// TIA Portal V20 program export: 6 tag tables, 4 data types, 72 data blocks, 38 code blocks (in call order from the OBs), 73 instance data blocks

VAR_GLOBAL   // PLC tag table "06_ProductionData"
END_VAR
VAR_GLOBAL CONSTANT   // user constants
   NO_DATASETS_CYCLETIMER : Int := 8;   // SICAR: Anzahl Datensätze Taktzeiten / SICAR: Number of data sets Cycle Timer
   NO_DATASETS_LIMITVALUES : Int := 1;   // SICAR: Anzahl Datensätze Grenzwerte / SICAR: Number of data sets Limit Value
   NO_DATASETS_SHIFTCOUNTER : Int := 1;   // SICAR: Anzahl Datensätze Schichtzähler / SICAR: Number of data sets Shift Counter
   NO_DATASETS_COUNTER : Int := 1;   // SICAR: Anzahl Datensätze Zähler / SICAR: Number of data sets Counter
END_VAR

VAR_GLOBAL   // PLC tag table "07_Energy"
   PAC3220InPut AT %I500.0 : "LER_typePAC3220Input_Status";
   "Active energy import tariff 1(F)" AT %ID612 : Real;
   "Reactive energy import tariff 1 (F)" AT %ID616 : Real;
   "Apparent energy tariff 1 (F)" AT %ID620 : Real;
   "Active energy export tariff 1(F)" AT %ID624 : Real;
   "Reactive energy export tariff 1 (F)" AT %ID628 : Real;
   "Apparent power L1" AT %ID632 : Real;
   "Apparent power L2" AT %ID636 : Real;
   "Apparent power L3" AT %ID640 : Real;
   "Active power L1" AT %ID644 : Real;
   "Active power L2" AT %ID648 : Real;
   "Active power L3" AT %ID652 : Real;
   "Reactive power L1" AT %ID656 : Real;
   "Reactive power L2" AT %ID660 : Real;
   "Reactive power L3" AT %ID664 : Real;
   PAC3220OutPut AT %Q500.0 : "LER_typePAC3220Output_Status";
END_VAR
VAR_GLOBAL CONSTANT   // user constants
   NO_OF_MACHINES : USInt := 1;   // SICAR: No of machines for EE-Monitor
   NO_OF_MEASUREPOINTS : USInt := 1;   // SICAR: Anzahl der Messstellen für EE-Monitor / SICAR: No of measurepoints for EE-Monitor
   "DP_FRWA1_1_0_000CC1-KE50~DP_FRWA1_1_0_000CC1-KE50_900" : Hw_Io := 10;
END_VAR

VAR_GLOBAL   // PLC tag table "08_CmInfo"
END_VAR
VAR_GLOBAL CONSTANT   // user constants
   NO_OF_RF_IDENT_DEVICES : USInt := 0;   // SICAR: Anzahl der RF Lesestellen / SICAR: Number of RF readers
   NO_OF_RF_ANTENNA_DEVICES : USInt := 2;   // SICAR: Number of RF antennas
END_VAR

VAR_GLOBAL   // PLC tag table "11_Settings"
END_VAR
VAR_GLOBAL CONSTANT   // user constants
   MAX_NO_OF_DEVICES_IRT : Int := 200;
   MAX_NO_OF_MODULES_IRT : Int := 200;
   MAX_NO_OF_DEVICES_RT : Int := 200;
   MAX_NO_OF_MODULES_RT : Int := 200;
END_VAR

VAR_GLOBAL   // PLC tag table "CentralFunctions"
END_VAR
VAR_GLOBAL CONSTANT   // user constants
   MAX_NO_OF_DEVICES_X1 : Int := 100;
   MAX_NO_OF_MODULES_X1 : Int := 100;
   MAX_NO_OF_DEVICES_X2 : Int := 100;
   MAX_NO_OF_MODULES_X2 : Int := 100;
END_VAR

VAR_GLOBAL   // PLC tag table "TextListId"
END_VAR
VAR_GLOBAL CONSTANT   // user constants
   TEXT_LIST_ID_PN_DEV_DIAG : Int := 591;   // SICAR: ID von SPS Alarm Textlist / SICAR: ID of PLC Alarm text list
   TEXT_LIST_ID_CHECKSUM : Int := 584;   // SICAR: ID von SPS Alarm Textlist / SICAR: ID of PLC Alarm text list
   TEXT_LIST_ID_EEEMONITOR_REPORT : Int := 562;   // SICAR: ID von SPS Alarm Textlist / SICAR: ID of PLC Alarm text list
   TEXT_LIST_ID_EEEMONITOR_CALC : Int := 561;   // SICAR: ID von SPS Alarm Textlist / SICAR: ID of PLC Alarm text list
   TEXT_LIST_ID_IDENT_SYSTEM : Int := 516;   // SICAR: ID of PLC Alarm for ident demo
   TEXT_LIST_ID_SMC_PD : Int := 585;   // SICAR: ID von SPS Alarm Textlist / SICAR: ID of PLC Alarm text list
   TEXT_LIST_ID_MOTORSTARTERS : Int := 588;   // SICAR: ID of PLC Alarm for motorstarter Demo
   TEXT_LIST_ID_DEV_FWD_REV : Int := 592;   // SICAR: ID of PLC Alarm for motorstarter Demo
END_VAR

TYPE "typeReelCutToStack"
   STRUCT
      Load_Enable : Bool;
      Load_Complete_Comfirm : Bool;
      Cell_Data_Report : Bool;
      signal3 : Bool;
      signal4 : Bool;
      signal5 : Bool;
      signal6 : Bool;
      signal7 : Bool;
      signal8 : Bool;
      signal9 : Bool;
      signal10 : Bool;
      signal11 : Bool;
      signal12 : Bool;
      signal13 : Bool;
      signal14 : Bool;
      HeartBeat : Bool;
      signal16 : Bool;
      signal17 : Bool;
      signal18 : Bool;
      signal19 : Bool;
      signal20 : Bool;
      signal21 : Bool;
      signal22 : Bool;
      signal23 : Bool;
      signal24 : Bool;
      signal25 : Bool;
      signal26 : Bool;
      signal27 : Bool;
      signal28 : Bool;
      signal29 : Bool;
      signal30 : Bool;
      signal31 : Bool;
      signal32 : Bool;
      signal33 : Bool;
      signal34 : Bool;
      signal35 : Bool;
      signal36 : Bool;
      signal37 : Bool;
      signal38 : Bool;
      signal39 : Bool;
      signal40 : Bool;
      signal41 : Bool;
      signal42 : Bool;
      signal43 : Bool;
      signal44 : Bool;
      signal45 : Bool;
      signal46 : Bool;
      signal47 : Bool;
      signal48 : Bool;
      signal49 : Bool;
      signal50 : Bool;
      signal51 : Bool;
      signal52 : Bool;
      signal53 : Bool;
      signal54 : Bool;
      signal55 : Bool;
      signal56 : Bool;
      signal57 : Bool;
      signal58 : Bool;
      signal59 : Bool;
      signal60 : Bool;
      signal61 : Bool;
      signal62 : Bool;
      signal63 : Bool;
      signal64 : Bool;
      signal65 : Bool;
      signal66 : Bool;
      signal67 : Bool;
      signal68 : Bool;
      signal69 : Bool;
      signal70 : Bool;
      signal71 : Bool;
      signal72 : Bool;
      signal73 : Bool;
      signal74 : Bool;
      signal75 : Bool;
      signal76 : Bool;
      signal77 : Bool;
      signal78 : Bool;
      signal79 : Bool;
      signal80 : Bool;
      signal81 : Bool;
      signal82 : Bool;
      signal83 : Bool;
      signal84 : Bool;
      signal85 : Bool;
      signal86 : Bool;
      signal87 : Bool;
      signal88 : Bool;
      signal89 : Bool;
      signal90 : Bool;
      signal91 : Bool;
      signal92 : Bool;
      signal93 : Bool;
      signal94 : Bool;
      signal95 : Bool;
   END_STRUCT;
END_TYPE

TYPE "typeStackToReelCut"
   STRUCT
      Load_Requset : Bool;
      Load_Busy : Bool;
      Load_Complete : Bool;
      Cell_Data_Request : Bool;
      Cell_Data_Report_Ack : Bool;
      Cell_Data_Report_Nck : Bool;
      signal6 : Bool;
      signal7 : Bool;
      signal8 : Bool;
      signal9 : Bool;
      signal10 : Bool;
      signal11 : Bool;
      signal12 : Bool;
      signal13 : Bool;
      signal14 : Bool;
      HeartBeat : Bool;
      signal16 : Bool;
      signal17 : Bool;
      signal18 : Bool;
      signal19 : Bool;
      signal20 : Bool;
      signal21 : Bool;
      signal22 : Bool;
      signal23 : Bool;
      signal24 : Bool;
      signal25 : Bool;
      signal26 : Bool;
      signal27 : Bool;
      signal28 : Bool;
      signal29 : Bool;
      signal30 : Bool;
      signal31 : Bool;
      signal32 : Bool;
      signal33 : Bool;
      signal34 : Bool;
      signal35 : Bool;
      signal36 : Bool;
      signal37 : Bool;
      signal38 : Bool;
      signal39 : Bool;
      signal40 : Bool;
      signal41 : Bool;
      signal42 : Bool;
      signal43 : Bool;
      signal44 : Bool;
      signal45 : Bool;
      signal46 : Bool;
      signal47 : Bool;
      signal48 : Bool;
      signal49 : Bool;
      signal50 : Bool;
      signal51 : Bool;
      signal52 : Bool;
      signal53 : Bool;
      signal54 : Bool;
      signal55 : Bool;
      signal56 : Bool;
      signal57 : Bool;
      signal58 : Bool;
      signal59 : Bool;
      signal60 : Bool;
      signal61 : Bool;
      signal62 : Bool;
      signal63 : Bool;
      signal64 : Bool;
      signal65 : Bool;
      signal66 : Bool;
      signal67 : Bool;
      signal68 : Bool;
      signal69 : Bool;
      signal70 : Bool;
      signal71 : Bool;
      signal72 : Bool;
      signal73 : Bool;
      signal74 : Bool;
      signal75 : Bool;
      signal76 : Bool;
      signal77 : Bool;
      signal78 : Bool;
      signal79 : Bool;
      signal80 : Bool;
      signal81 : Bool;
      signal82 : Bool;
      signal83 : Bool;
      signal84 : Bool;
      signal85 : Bool;
      signal86 : Bool;
      signal87 : Bool;
      signal88 : Bool;
      signal89 : Bool;
      signal90 : Bool;
      signal91 : Bool;
      signal92 : Bool;
      signal93 : Bool;
      signal94 : Bool;
      signal95 : Bool;
   END_STRUCT;
END_TYPE

TYPE "typeIdentRf"
// stored: Access Published
   STRUCT
      IdentRfAntena : Array[0.."NO_OF_RF_ANTENNA_DEVICES"] of "LSicar_typeIdentInterfaceHmi";
   END_STRUCT;
END_TYPE

TYPE "typeIdentRfHmi"
// stored: Access Published
   STRUCT
      selectedRfReader : USInt;   // Reader ID
      selectedAntena : USInt;
      rfReaderId : USInt;   // RF Reader ID
      numberOfRf : USInt;   // Anzahl der RFID Antriebe / Number of used RFIDs
      rfReader : "LSicar_typeIdentInterfaceHmi";   // RF Reader
   END_STRUCT;
END_TYPE

DATA_BLOCK "Hmi"   // DB4
// stored: MemoryReserve 100
   VAR
      mainHeader : Array[0.."NO_OF_PANELS"] of "LAF_typeHeader";   // Input from the status bar of the HMI
      operationInterlock : "LAF_typeOperationInterlockInterface";
   END_VAR
BEGIN
   mainHeader[0].plcToHmi.modeRequestsButtons.visibility := 16#0;
   mainHeader[0].plcToHmi.specialFunctionButtons.visibility := 16#0071_FFFF;
   mainHeader[0].plcToHmi.specialFunctionButtons.operatorControlAllowed := 16#0;
   mainHeader[0].plcToHmi.specialFunctionButtons.active := 16#0;
END_DATA_BLOCK

DATA_BLOCK "LRemoteAccess_Data"   // DB275
TITLE = Data
AUTHOR : Siemens
// Storing data about mobile panel and UCP connection status
// stored: MemoryReserve 100
   VAR
      mobilePanel1 : "LRemoteAccess_typeMobilePanel";
      connectionBoxes : Array[1..2] of "LRemoteAccess_typeConnectionBox";
      ActivationMobileDP { S7_SetPoint := 'True'} : "LRemoteAccess_typeMobile_DeActivate";   // Activate Mobile Panel
      DeactivationMobileDP { S7_SetPoint := 'True'} : "LRemoteAccess_typeMobile_DeActivate";   // Deactivate Mobile Panel
      connectionTimeout { S7_SetPoint := 'True'} : Time := T#5s;   // Connection timeout. Keep greater than 3 sec. Default 5 sec.
   END_VAR
BEGIN
   connectionBoxes[1].ID := 14;
   connectionBoxes[2].ID := 15;
END_DATA_BLOCK

DATA_BLOCK "Simulation"   // DB134
TITLE = Simulation
// Simulation data
// stored: MemoryReserve 100
   VAR
      data : "LAF_typeSimulation";
      hmiSimulationAxis { S7_SetPoint := 'True'} : Array[0..10] of LReal;
   END_VAR
BEGIN
END_DATA_BLOCK

DATA_BLOCK "HMI_Interface_Overview"   // DB276
// stored: Access Published, MemoryReserve 100
   VAR
      State : Struct
         "Anode Reel Cut" : "HMI_IF_OverView_Unit_UDT";
         "Cathode Reel Cut" : "HMI_IF_OverView_Unit_UDT";
         "Stacker #1" : "HMI_IF_OverView_Unit_UDT";
         "Stacker #2" : "HMI_IF_OverView_Unit_UDT";
         Inspection : "HMI_IF_OverView_Unit_UDT";
      END_STRUCT;
   END_VAR
BEGIN
END_DATA_BLOCK

DATA_BLOCK "LAF_InternalManual"   // DB43
VERSION : 19.0
// stored: MemoryReserve 100
   VAR
      hmi : Array[1..1] of "LAF_typeManHmiDisp";   // Anzahl der HMIs - modifizieren Sie die Array-Größe auf Basis der erforderlichen HMI / number of HMIs - modify the array size based on the required HMIs / número de HMI: modificar el tamaño del array según las HMI requeridas / nombre d'IHM - modifier la taille du tableau en fonction du nombre d'IHM requis / numero di HMI - modificare la dimensione di array in base alle HMI richieste / HMI 수 - 필요한 HMI에 따라 배열 크기를 수정합니다. / HMI 数量 - 根据所需的 HMI 修改数组大小
      manualOperationEnabled : Bool;   // feedback whether the manual operation lines are selected
      emsWithManualOpConfigured { ExternalWritable := 'False'} : "LGM_emsWithManualOpConfigured";   // List of EMs with manual operation configured, for HMI button visibility
      disableUnit1 { S7_SetPoint := 'True'} : Bool;
      RisingEdge : Bool;
   END_VAR
BEGIN
END_DATA_BLOCK

DATA_BLOCK "ManualOperationControl_Template"   // DB91
// stored: MemoryReserve 100
   VAR
      manualOperationEm { ExternalAccessible := 'False'; ExternalVisible := 'False'; ExternalWritable := 'False'} : "LAF_typeManEm";
      manualOperationEmArea { ExternalAccessible := 'False'; ExternalVisible := 'False'; ExternalWritable := 'False'} : Array[1..1] of "LAF_typeManOperationArea";
      manualOperationCms { ExternalAccessible := 'False'; ExternalVisible := 'False'; ExternalWritable := 'False'} : Array[1..1] of "LAF_typeManOperation";
   END_VAR
BEGIN
   manualOperationEm.equipmentModuleNum := 3400;
END_DATA_BLOCK

DATA_BLOCK "OperatorPrompts"   // DB123
// stored: Access Published, MemoryReserve 100
   VAR
      triggers { ExternalAccessible := 'False'; ExternalVisible := 'False'; ExternalWritable := 'False'} : Array[1..63] of Bool;
      activeOperatorPrompt { ExternalWritable := 'False'} : Int;
      ack : Bool;
   END_VAR
BEGIN
END_DATA_BLOCK

DATA_BLOCK "ProdDataInterfaceHmi"   // DB53
TITLE = HMI und Anwender Schnittstelle für Produktionsdaten / HMI and user interface for production data
AUTHOR : SICAR
FAMILY : ProdData
// FUNKTIONSBESCHREIBUNG: 
// Der Baustein beinhaltet alle Informationen zum und vom HMI, sowie die Anwenderschnittstellen für die Produktionsdaten
// Weitere Hinweise: siehe SICAR anwenderdefinierte Dokumentation / SICAR Online-Hilfe.
// DESCRIPTION OF FUNCTIONS:
// stored: MemoryReserve 100
   VAR RETAIN
      numberOfDataSets : "LSicar_typeNumberOfDataSets";   // Anzahl konfigurierter Datensätze / Number of configured data sets
   END_VAR
   VAR
      colorCodeLimitSummary : UInt;   // Gesamt Status Grenzwerte / Overall status Limit values
      colorCodeLimitSelButton : Array[0..8] of UInt;   // Farbcode für Datensatz Anwahl Button (Grenzwerte) / Color code for data set select button (Limit values)
   END_VAR
   VAR RETAIN
      counterDataSetSel : Int := 1;   // Angewählter Datensatz Zaehler / selected data set counter
      counterDataSet : Array[0.."NO_DATASETS_COUNTER"] of "LSicar_typeCounter";   // Datensätze Zähler / Data sets counter
      cycleTimerDataSetSel : Int := 1;   // Angewaehlter Datensatz Taktzeiten / selected data set cycle timer
      cycleTimerDataSet : Array[0.."NO_DATASETS_CYCLETIMER"] of "LSicar_typeCycleTimer";   // Datensätze Taktzeiten / Data sets cycle timer
      limitValueDataSetSel : Int := 1;   // Angwaehlter Datensatz Grenzwerte / selected data set limit values
      limitDataSet : Array[0.."NO_DATASETS_LIMITVALUES"] of "LSicar_typeLimitValue";   // Datensätze Grenzwerte / Data sets limit .values
      shiftCounterDataSetSel : Int := 1;   // Angewaehlter Datensatz Schichtzaehler / selected data set shift counter
      shiftCounterDataSet : Array[0.."NO_DATASETS_SHIFTCOUNTER"] of "LSicar_typeShiftCounter";   // Datensätze Schichtzähler / Data sets shift counter
      shiftCountOeeDataSetSel : Int := 1;   // Angewaehlter Datensatz OEE / selected data set OEE
      shiftCounterOeeDataSet : Array[0.."NO_DATASETS_SHIFTCOUNTER"] of "LSicar_typeShiftCounterOee";   // Datensätze Schichtzähler OEE / Data sets shift counter OEE
   END_VAR
BEGIN
END_DATA_BLOCK

DATA_BLOCK "ProdDataSimulation"   // DB5
{ DB_Accessible_From_OPC_UA := 'FALSE' }
// stored: DBAccessibleFromOPCUA false, DBAccessibleFromWebserver false, MemoryReserve 100
   VAR
      ProdDataCounter { ExternalAccessible := 'False'; ExternalVisible := 'False'; ExternalWritable := 'False'} : Struct   // Test tag prod data
         ProdDataCounter1Up1 : Bool;   // Test Variable Prod. Daten / Test tag prod data
         ProdDataCounter1Up2 : Bool;   // Test Variable Prod. Daten / Test tag prod data
         ProdDataCounter1Down1 : Bool;   // Test Variable Prod. Daten / Test tag prod data
         ProdDataCounter1Down2 : Bool;   // Test Variable Prod. Daten / Test tag prod data
         ProdDataCounter1Reset1 : Bool;   // Test Variable Prod. Daten / Test tag prod data
         ProdDataCounter1Reset2 : Bool;   // Test Variable Prod. Daten / Test tag prod data
         ProdDataCounter1ResetAll : Bool;   // Test Variable Prod. Daten / Test tag prod data
         ProdDataCounter2Up1 : Bool;
         ProdDataCounter2Up2 : Bool;
         ProdDataCounter2Down1 : Bool;
         ProdDataCounter2Down2 : Bool;
         ProdDataCounter2Reset1 : Bool;
         ProdDataCounter2Reset2 : Bool;
         ProdDataCounter2ResetAll : Bool;
         userInterfaceVisibilityDataSet1Counter : DWord := 2#0000_0000_0000_0000_0000_0000_0011_1111;
         userInterfaceVisibilityDataSet2Counter : DWord := 2#0000_0000_0000_1111_1111_1111_1111_1111;
         ProdDataEnable : Bool;
      END_STRUCT;
      ProdDataCyclic { ExternalAccessible := 'False'; ExternalVisible := 'False'; ExternalWritable := 'False'} : Struct   // Test tag prod data
         cycleTimer1Run1 : Bool;   // Test Variable Prod. Daten / Test tag prod data
         cycleTimer1Run2 : Bool;   // Test Variable Prod. Daten / Test tag prod data
         cycleTimer1Hold1 : Bool;   // Test Variable Prod. Daten / Test tag prod data
         cycleTimer1Hold2 : Bool;   // Test Variable Prod. Daten / Test tag prod data
         cycleTimer1Reset1 : Bool;   // Test Variable Prod. Daten / Test tag prod data
         cycleTimer1Reset2 : Bool;   // Test Variable Prod. Daten / Test tag prod data
         cycleTimer1ResetAll : Bool;   // Test Variable Prod. Daten / Test tag prod data
         cycleTimer2Run1 : Bool;   // Test Variable Prod. Daten / Test tag prod data
         cycleTimer2Run2 : Bool;   // Test Variable Prod. Daten / Test tag prod data
         cycleTimer2Hold1 : Bool;   // Test Variable Prod. Daten / Test tag prod data
         cycleTimer2Hold2 : Bool;   // Test Variable Prod. Daten / Test tag prod data
         cycleTimer2Reset1 : Bool;   // Test Variable Prod. Daten / Test tag prod data
         cycleTimer2Reset2 : Bool;   // Test Variable Prod. Daten / Test tag prod data
         cycleTimer2ResetAll : Bool;   // Test Variable Prod. Daten / Test tag prod data
         cyclicTimerEnable : Bool;
         userInterfaceVisibilityDataSet1Cyclic : DWord := 2#0000_0000_0000_0000_0000_0000_0000_1111;
         userInterfaceVisibilityDataSet2Cyclic : DWord := 2#0000_0000_0000_0000_0000_0000_0000_1111;
         userInterfaceVisibilityDataSet3Cyclic : DWord := 2#0000_0000_0000_1000_0111_1111_1101_1111;
         userInterfaceVisibilityDataSet4Cyclic : DWord := 2#0000_0000_0000_0000_0000_0000_1111_1111;
         userInterfaceVisibilityDataSet5Cyclic : DWord := 2#0000_0000_0000_0000_0000_0000_0000_0001;
         userInterfaceVisibilityDataSet6Cyclic : DWord := 2#0000_0000_0000_0000_0000_0000_0000_0111;
         userInterfaceVisibilityDataSet7Cyclic : DWord := 2#0000_0000_0000_0000_0011_1100_0000_0111;
         userInterfaceVisibilityDataSet8Cyclic : DWord := 2#0000_0000_0000_1111_1111_1100_1111_1111;
      END_STRUCT;
      ProdDataLimitValues { ExternalAccessible := 'False'; ExternalVisible := 'False'; ExternalWritable := 'False'} : Struct   // Test tag prod data
         limitVal1Count1PreWarn1 : Bool;   // Test Variable Prod. Daten / Test tag prod data
         limitVal1Count1PreWarn3 : Bool;   // Test Variable Prod. Daten / Test tag prod data
         limitVal1Count1PreWarn2 : Bool;   // Test Variable Prod. Daten / Test tag prod data
         limitVal1Count1Alarm1 : Bool;   // Test Variable Prod. Daten / Test tag prod data
         limitVal1Count1Alarm3 : Bool;   // Test Variable Prod. Daten / Test tag prod data
         limitVal1Count1Alarm2 : Bool;   // Test Variable Prod. Daten / Test tag prod data
         limitVal1Count1 : Bool;   // Test Variable Prod. Daten / Test tag prod data
         limitVal1Count2 : Bool;   // Test Variable Prod. Daten / Test tag prod data
         limitVal1Count3 : Bool;   // Test Variable Prod. Daten / Test tag prod data
         limitVal1Set1 : Bool;   // Test Variable Prod. Daten / Test tag prod data
         limitVal1Set3 : Bool;   // Test Variable Prod. Daten / Test tag prod data
         limitVal1Set2 : Bool;   // Test Variable Prod. Daten / Test tag prod data
         limitValuesEnable : Bool;
         userInterfaceVisibilityDataSet2LimitValues : DWord := 2#0000_0000_0000_0000_0000_0011_1111_1111;
         userInterfaceVisibilityDataSet1LimitValues : DWord := 2#0000_0000_0000_0000_0000_0000_0000_1111;
      END_STRUCT;
      ProdDataShiftCounter { ExternalAccessible := 'False'; ExternalVisible := 'False'; ExternalWritable := 'False'} : Struct   // Test tag prod data
         shiftCounter1Cnt1Curr : Bool;   // Test Variable Prod. Daten / Test tag prod data
         shiftCounter1Cnt1CurrOk : Bool;   // Test Variable Prod. Daten / Test tag prod data
         shiftCounter1Cnt2Curr : Bool;   // Test Variable Prod. Daten / Test tag prod data
         shiftCounter1Cnt2CurrOk : Bool;   // Test Variable Prod. Daten / Test tag prod data
         shiftCounter1Cnt3Curr : Bool;   // Test Variable Prod. Daten / Test tag prod data
         shiftCounter1Cnt3CurrOk : Bool;   // Test Variable Prod. Daten / Test tag prod data
         shiftCounter1ResetAllExt : Bool;   // Test Variable Prod. Daten / Test tag prod data
         ShiftCounterEnable : Bool;
         userInterfaceVisibilityDataSet2ShiftCounter : DWord := 2#0000_0000_0000_0000_0000_0011_1111_1111;
         userInterfaceVisibilityDataSet1ShiftCounter : DWord := 2#0000_0000_0000_0000_0000_0000_0000_1111;
      END_STRUCT;
      ProdDataShiftCounterOEE { ExternalAccessible := 'False'; ExternalVisible := 'False'; ExternalWritable := 'False'} : Struct   // Test tag prod data
         ShiftCounterOEEEnable : Bool;
         userInterfaceVisibilityDataSet2ShiftCounterOEE : DWord := 2#0000_0000_0000_0000_0000_0011_1111_1111;
         userInterfaceVisibilityDataSet1ShiftCounterOEE : DWord := 2#0000_0000_0000_0000_0000_0000_0000_1111;
      END_STRUCT;
   END_VAR
BEGIN
END_DATA_BLOCK

DATA_BLOCK "ShiftInitBools"   // DB257
// stored: MemoryReserve 100
   VAR
      earlyShift : Bool;
      lateShift : Bool;
      nightShift : Bool;
   END_VAR
BEGIN
END_DATA_BLOCK

DATA_BLOCK "ShiftTimesList"   // DB52
TITLE = Shifttimes / Shift times
{ DB_Accessible_From_OPC_UA := 'FALSE' }
AUTHOR : SICAR
FAMILY : Shiftmodel
// Schichtzeiten Liste / Shift times List
// stored: DBAccessibleFromOPCUA false, MemoryReserve 100
   VAR
      list { ExternalAccessible := 'False'; ExternalVisible := 'False'; ExternalWritable := 'False'} : Array[0..10] of "LSicar_typeShiftmodTime1DaySel";   // Schichtmodel Liste / Shiftmodel list
   END_VAR
BEGIN
   list[3].listValidFor.sunday := TRUE;
   list[4].listValidFor.sunday := FALSE;
   list[1..3].listValidFor.monday := TRUE;
   list[4].listValidFor.monday := FALSE;
   list[1..3].listValidFor.tuesday := TRUE;
   list[4].listValidFor.tuesday := FALSE;
   list[1..3].listValidFor.wednesday := TRUE;
   list[4].listValidFor.wednesday := FALSE;
   list[1..3].listValidFor.thursday := TRUE;
   list[4].listValidFor.thursday := FALSE;
   list[1].listValidFor.friday := TRUE;
   list[3].listValidFor.friday := TRUE;
   list[4].listValidFor.friday := FALSE;
   list[3].listValidFor.saturday := TRUE;
   list[4].listValidFor.saturday := FALSE;
   list[1].shift[1].endCircuitTime := TOD#05:57:00;
   list[1].shift[2].endCircuitTime := TOD#13:57:00;
   list[1].shift[3].endCircuitTime := TOD#21:57:00;
   list[2].shift[1].endCircuitTime := TOD#04:57:00;
   list[2].shift[2].endCircuitTime := TOD#14:27:00;
   list[3].shift[1].endCircuitTime := TOD#05:57:00;
   list[3].shift[2].endCircuitTime := TOD#14:27:00;
   list[3].shift[3].endCircuitTime := TOD#22:57:00;
   list[4].shift[1..3].endCircuitTime := TOD#00:00:00;
   list[1].shift[1].start := TOD#06:00:00;
   list[1].shift[2].start := TOD#14:00:00;
   list[1].shift[3].start := TOD#22:00:00;
   list[2].shift[1].start := TOD#05:00:00;
   list[2].shift[2].start := TOD#14:30:00;
   list[3].shift[1].start := TOD#06:00:00;
   list[3].shift[2].start := TOD#14:30:00;
   list[3].shift[3].start := TOD#23:00:00;
   list[4].shift[1..3].start := TOD#00:00:00;
   list[1].shift[1].break[1].start := TOD#08:00:00;
   list[1].shift[1].break[2].start := TOD#10:00:00;
   list[1].shift[1].break[3].start := TOD#12:00:00;
   list[1].shift[1].break[4].start := TOD#00:00:00;
   list[1].shift[2].break[1].start := TOD#16:00:00;
   list[1].shift[2].break[2].start := TOD#18:00:00;
   list[1].shift[2].break[3].start := TOD#20:00:00;
   list[1].shift[3].break[1].start := TOD#00:00:00;
   list[1].shift[3].break[2].start := TOD#02:00:00;
   list[1].shift[3].break[3].start := TOD#04:00:00;
   list[2].shift[1].break[1].start := TOD#07:00:00;
   list[2].shift[1].break[2].start := TOD#09:00:00;
   list[2].shift[1].break[3].start := TOD#11:00:00;
   list[2].shift[1].break[4].start := TOD#13:00:00;
   list[2].shift[2].break[1].start := TOD#16:30:00;
   list[2].shift[2].break[2].start := TOD#18:30:00;
   list[2].shift[2].break[3].start := TOD#20:30:00;
   list[2].shift[2].break[4].start := TOD#22:00:00;
   list[3].shift[1].break[1].start := TOD#08:00:00;
   list[3].shift[1].break[2].start := TOD#10:00:00;
   list[3].shift[1].break[3].start := TOD#11:30:00;
   list[3].shift[1].break[4].start := TOD#12:30:00;
   list[3].shift[2].break[1].start := TOD#16:00:00;
   list[3].shift[2].break[2].start := TOD#18:00:00;
   list[3].shift[2].break[3].start := TOD#19:30:00;
   list[3].shift[2].break[4].start := TOD#20:30:00;
   list[3].shift[3].break[1].start := TOD#00:00:00;
   list[3].shift[3].break[2].start := TOD#02:00:00;
   list[3].shift[3].break[3].start := TOD#03:30:00;
   list[3].shift[3].break[4].start := TOD#04:30:00;
   list[4].shift[1].break[1..4].start := TOD#00:00:00;
   list[4].shift[2].break[1..4].start := TOD#00:00:00;
   list[4].shift[3].break[1..4].start := TOD#00:00:00;
   list[1].shift[1].break[1].startCircuitTime := TOD#08:02:00;
   list[1].shift[1].break[2].startCircuitTime := TOD#00:00:00;
   list[1].shift[1].break[3].startCircuitTime := TOD#12:02:00;
   list[1].shift[1].break[4].startCircuitTime := TOD#00:00:00;
   list[1].shift[2].break[1].startCircuitTime := TOD#16:02:00;
   list[1].shift[2].break[2].startCircuitTime := TOD#00:00:00;
   list[1].shift[2].break[3].startCircuitTime := TOD#20:02:00;
   list[1].shift[3].break[1].startCircuitTime := TOD#00:02:00;
   list[1].shift[3].break[2].startCircuitTime := TOD#00:00:00;
   list[1].shift[3].break[3].startCircuitTime := TOD#04:02:00;
   list[2].shift[1].break[1].startCircuitTime := TOD#07:02:00;
   list[2].shift[1].break[2].startCircuitTime := TOD#00:00:00;
   list[2].shift[1].break[3].startCircuitTime := TOD#11:02:00;
   list[2].shift[1].break[4].startCircuitTime := TOD#13:02:00;
   list[2].shift[2].break[1].startCircuitTime := TOD#16:32:00;
   list[2].shift[2].break[2].startCircuitTime := TOD#00:00:00;
   list[2].shift[2].break[3].startCircuitTime := TOD#20:32:00;
   list[2].shift[2].break[4].startCircuitTime := TOD#22:02:00;
   list[3].shift[1].break[1].startCircuitTime := TOD#00:00:00;
   list[3].shift[1].break[2].startCircuitTime := TOD#10:02:00;
   list[3].shift[1].break[3].startCircuitTime := TOD#00:00:00;
   list[3].shift[1].break[4].startCircuitTime := TOD#12:32:00;
   list[3].shift[2].break[1].startCircuitTime := TOD#00:00:00;
   list[3].shift[2].break[2].startCircuitTime := TOD#18:02:00;
   list[3].shift[2].break[3].startCircuitTime := TOD#00:00:00;
   list[3].shift[2].break[4].startCircuitTime := TOD#20:32:00;
   list[3].shift[3].break[1].startCircuitTime := TOD#00:00:00;
   list[3].shift[3].break[2].startCircuitTime := TOD#02:02:00;
   list[3].shift[3].break[3..4].startCircuitTime := TOD#00:00:00;
   list[4].shift[1].break[1..4].startCircuitTime := TOD#00:00:00;
   list[4].shift[2].break[1..4].startCircuitTime := TOD#00:00:00;
   list[4].shift[3].break[1..4].startCircuitTime := TOD#00:00:00;
   list[1].shift[1].break[1].endCircuitTime := TOD#08:13:00;
   list[1].shift[1].break[2].endCircuitTime := TOD#00:00:00;
   list[1].shift[1].break[3].endCircuitTime := TOD#12:13:00;
   list[1].shift[1].break[4].endCircuitTime := TOD#00:00:00;
   list[1].shift[2].break[1].endCircuitTime := TOD#16:13:00;
   list[1].shift[2].break[2].endCircuitTime := TOD#00:00:00;
   list[1].shift[2].break[3].endCircuitTime := TOD#20:13:00;
   list[1].shift[3].break[1].endCircuitTime := TOD#00:13:00;
   list[1].shift[3].break[2].endCircuitTime := TOD#00:00:00;
   list[1].shift[3].break[3].endCircuitTime := TOD#04:13:00;
   list[2].shift[1].break[1].endCircuitTime := TOD#07:13:00;
   list[2].shift[1].break[2].endCircuitTime := TOD#00:00:00;
   list[2].shift[1].break[3].endCircuitTime := TOD#11:13:00;
   list[2].shift[1].break[4].endCircuitTime := TOD#13:13:00;
   list[2].shift[2].break[1].endCircuitTime := TOD#16:43:00;
   list[2].shift[2].break[2].endCircuitTime := TOD#00:00:00;
   list[2].shift[2].break[3].endCircuitTime := TOD#20:43:00;
   list[2].shift[2].break[4].endCircuitTime := TOD#22:13:00;
   list[3].shift[1].break[1].endCircuitTime := TOD#00:00:00;
   list[3].shift[1].break[2].endCircuitTime := TOD#10:13:00;
   list[3].shift[1].break[3].endCircuitTime := TOD#00:00:00;
   list[3].shift[1].break[4].endCircuitTime := TOD#12:43:00;
   list[3].shift[2].break[1].endCircuitTime := TOD#00:00:00;
   list[3].shift[2].break[2].endCircuitTime := TOD#18:13:00;
   list[3].shift[2].break[3].endCircuitTime := TOD#00:00:00;
   list[3].shift[2].break[4].endCircuitTime := TOD#20:43:00;
   list[3].shift[3].break[1].endCircuitTime := TOD#00:00:00;
   list[3].shift[3].break[2].endCircuitTime := TOD#02:13:00;
   list[3].shift[3].break[3..4].endCircuitTime := TOD#00:00:00;
   list[4].shift[1].break[1..4].endCircuitTime := TOD#00:00:00;
   list[4].shift[2].break[1..4].endCircuitTime := TOD#00:00:00;
   list[4].shift[3].break[1..4].endCircuitTime := TOD#00:00:00;
   list[1].shift[1].break[1].end := TOD#08:15:00;
   list[1].shift[1].break[2].end := TOD#10:10:00;
   list[1].shift[1].break[3].end := TOD#12:15:00;
   list[1].shift[1].break[4].end := TOD#00:00:00;
   list[1].shift[2].break[1].end := TOD#16:15:00;
   list[1].shift[2].break[2].end := TOD#18:10:00;
   list[1].shift[2].break[3].end := TOD#20:15:00;
   list[1].shift[3].break[1].end := TOD#00:15:00;
   list[1].shift[3].break[2].end := TOD#02:10:00;
   list[1].shift[3].break[3].end := TOD#04:15:00;
   list[2].shift[1].break[1].end := TOD#07:15:00;
   list[2].shift[1].break[2].end := TOD#09:10:00;
   list[2].shift[1].break[3].end := TOD#11:15:00;
   list[2].shift[1].break[4].end := TOD#13:15:00;
   list[2].shift[2].break[1].end := TOD#16:45:00;
   list[2].shift[2].break[2].end := TOD#18:40:00;
   list[2].shift[2].break[3].end := TOD#20:45:00;
   list[2].shift[2].break[4].end := TOD#22:15:00;
   list[3].shift[1].break[1].end := TOD#08:10:00;
   list[3].shift[1].break[2].end := TOD#10:15:00;
   list[3].shift[1].break[3].end := TOD#11:40:00;
   list[3].shift[1].break[4].end := TOD#12:45:00;
   list[3].shift[2].break[1].end := TOD#16:10:00;
   list[3].shift[2].break[2].end := TOD#18:15:00;
   list[3].shift[2].break[3].end := TOD#19:40:00;
   list[3].shift[2].break[4].end := TOD#20:45:00;
   list[3].shift[3].break[1].end := TOD#00:10:00;
   list[3].shift[3].break[2].end := TOD#02:15:00;
   list[3].shift[3].break[3].end := TOD#03:40:00;
   list[3].shift[3].break[4].end := TOD#04:45:00;
   list[4].shift[1].break[1..4].end := TOD#00:00:00;
   list[4].shift[2].break[1..4].end := TOD#00:00:00;
   list[4].shift[3].break[1..4].end := TOD#00:00:00;
   list[1].shift[1].end := TOD#13:30:00;
   list[1].shift[2].end := TOD#21:30:00;
   list[1].shift[3].end := TOD#05:30:00;
   list[2].shift[1].end := TOD#14:00:00;
   list[2].shift[2].end := TOD#23:30:00;
   list[3].shift[1].end := TOD#13:30:00;
   list[3].shift[2].end := TOD#21:30:00;
   list[3].shift[3].end := TOD#05:30:00;
   list[4].shift[1..3].end := TOD#00:00:00;
   list[1].shift[1].startCircuitTime := TOD#13:33:00;
   list[1].shift[2].startCircuitTime := TOD#21:33:00;
   list[1].shift[3].startCircuitTime := TOD#05:33:00;
   list[2].shift[1].startCircuitTime := TOD#14:03:00;
   list[2].shift[2].startCircuitTime := TOD#23:33:00;
   list[3].shift[1].startCircuitTime := TOD#13:33:00;
   list[3].shift[2].startCircuitTime := TOD#21:33:00;
   list[3].shift[3].startCircuitTime := TOD#05:33:00;
   list[4].shift[1..3].startCircuitTime := TOD#00:00:00;
END_DATA_BLOCK

DATA_BLOCK "Settings"   // DB6
{ DB_Accessible_From_OPC_UA := 'FALSE' }
// stored: Access Published, DBAccessibleFromOPCUA false, DBAccessibleFromWebserver false, MemoryReserve 100
   VAR
      diagPlc : "LAF_typePlcDiag";   // HMI Schnittstelle PLC Diagnose / HMI interface PLC diag
      checksum : "LAF_typeChecksum";   // HMI Schnittstelle PLCChecksum / HMI interface PLCChecksum
      diagMemCard : "LAF_typeMemCardDiag";   // HMI Schnittstelle SMCDiag / HMI interface SMCDiag
      cycleTimes : "LSicar_typeGlobalRuntime";
      setLocalPlcTime : "LAF_typeSetPlcTime";
      ITConnection : Bool := FALSE;   // Provides a visual representation of the connection with the IT systems.
   END_VAR
BEGIN
END_DATA_BLOCK

DATA_BLOCK "ManualOperationControl_U1Em0"   // DB104
// stored: MemoryReserve 100
   VAR
      manualOperationEm { ExternalAccessible := 'False'; ExternalVisible := 'False'; ExternalWritable := 'False'} : "LAF_typeManEm";
      manualOperationEmArea { ExternalAccessible := 'False'; ExternalVisible := 'False'; ExternalWritable := 'False'} : Array[1..2] of "LAF_typeManOperationArea";
      manualOperationCms { ExternalAccessible := 'False'; ExternalVisible := 'False'; ExternalWritable := 'False'} : Array[1..45] of "LAF_typeManOperation";
      axis { ExternalAccessible := 'False'; ExternalVisible := 'False'; ExternalWritable := 'False'} : Array[0..1] of "LBC_typeAxisControlInterface";
      axis64Pos { ExternalAccessible := 'False'; ExternalVisible := 'False'; ExternalWritable := 'False'} : Array[0..0] of "LBC_typeAxis64PosInterface";
      softCam { ExternalAccessible := 'False'; ExternalVisible := 'False'; ExternalWritable := 'False'} : Array[0..1] of "LER_typeSoftCamRelation";
      sina { ExternalAccessible := 'False'; ExternalVisible := 'False'; ExternalWritable := 'False'} : Array[0..0] of "LBC_typeSinaSpeedInterface";
      twoWayActuator { ExternalAccessible := 'False'; ExternalVisible := 'False'; ExternalWritable := 'False'} : Array[0..2] of "LBC_typeTwoWayActuatorInterface";
   END_VAR
BEGIN
   manualOperationEm.equipmentModuleNum := 1010;
END_DATA_BLOCK

DATA_BLOCK "ManualOperationControl_U1Em1"   // DB156
// stored: MemoryReserve 100
   VAR
      manualOperationEm { ExternalAccessible := 'False'; ExternalVisible := 'False'; ExternalWritable := 'False'} : "LAF_typeManEm";
      manualOperationEmArea { ExternalAccessible := 'False'; ExternalVisible := 'False'; ExternalWritable := 'False'} : Array[1..2] of "LAF_typeManOperationArea";
      manualOperationCms { ExternalAccessible := 'False'; ExternalVisible := 'False'; ExternalWritable := 'False'} : Array[1..45] of "LAF_typeManOperation";
      axis { ExternalAccessible := 'False'; ExternalVisible := 'False'; ExternalWritable := 'False'} : Array[0..1] of "LBC_typeAxisControlInterface";
      axis64Pos { ExternalAccessible := 'False'; ExternalVisible := 'False'; ExternalWritable := 'False'} : Array[0..0] of "LBC_typeAxis64PosInterface";
      softCam { ExternalAccessible := 'False'; ExternalVisible := 'False'; ExternalWritable := 'False'} : Array[0..1] of "LER_typeSoftCamRelation";
      sina { ExternalAccessible := 'False'; ExternalVisible := 'False'; ExternalWritable := 'False'} : Array[0..0] of "LBC_typeSinaSpeedInterface";
      twoWayActuator { ExternalAccessible := 'False'; ExternalVisible := 'False'; ExternalWritable := 'False'} : Array[0..2] of "LBC_typeTwoWayActuatorInterface";
   END_VAR
BEGIN
   manualOperationEm.equipmentModuleNum := 1020;
END_DATA_BLOCK

DATA_BLOCK "ManualOperationControl_U1Em2"   // DB144
// stored: MemoryReserve 100
   VAR
      manualOperationEm { ExternalAccessible := 'False'; ExternalVisible := 'False'; ExternalWritable := 'False'} : "LAF_typeManEm";
      manualOperationEmArea { ExternalAccessible := 'False'; ExternalVisible := 'False'; ExternalWritable := 'False'} : Array[1..2] of "LAF_typeManOperationArea";
      manualOperationCms { ExternalAccessible := 'False'; ExternalVisible := 'False'; ExternalWritable := 'False'} : Array[1..45] of "LAF_typeManOperation";
      axis { ExternalAccessible := 'False'; ExternalVisible := 'False'; ExternalWritable := 'False'} : Array[0..0] of "LBC_typeAxisControlInterface";
      axis64Pos { ExternalAccessible := 'False'; ExternalVisible := 'False'; ExternalWritable := 'False'} : Array[0..0] of "LBC_typeAxis64PosInterface";
      softCam { ExternalAccessible := 'False'; ExternalVisible := 'False'; ExternalWritable := 'False'} : Array[0..0] of "LER_typeSoftCamRelation";
      sina { ExternalAccessible := 'False'; ExternalVisible := 'False'; ExternalWritable := 'False'} : Array[0..0] of "LBC_typeSinaSpeedInterface";
      twoWayActuator { ExternalAccessible := 'False'; ExternalVisible := 'False'; ExternalWritable := 'False'} : Array[0..22] of "LBC_typeTwoWayActuatorInterface";
   END_VAR
BEGIN
   manualOperationEm.equipmentModuleNum := 1030;
END_DATA_BLOCK

DATA_BLOCK "ManualOperationControl_U1Em3"   // DB142
// stored: MemoryReserve 100
   VAR
      manualOperationEm { ExternalAccessible := 'False'; ExternalVisible := 'False'; ExternalWritable := 'False'} : "LAF_typeManEm";
      manualOperationEmArea { ExternalAccessible := 'False'; ExternalVisible := 'False'; ExternalWritable := 'False'} : Array[1..2] of "LAF_typeManOperationArea";
      manualOperationCms { ExternalAccessible := 'False'; ExternalVisible := 'False'; ExternalWritable := 'False'} : Array[1..45] of "LAF_typeManOperation";
      axis { ExternalAccessible := 'False'; ExternalVisible := 'False'; ExternalWritable := 'False'} : Array[0..0] of "LBC_typeAxisControlInterface";
      axis64Pos { ExternalAccessible := 'False'; ExternalVisible := 'False'; ExternalWritable := 'False'} : Array[0..0] of "LBC_typeAxis64PosInterface";
      softCam { ExternalAccessible := 'False'; ExternalVisible := 'False'; ExternalWritable := 'False'} : Array[0..0] of "LER_typeSoftCamRelation";
      sina { ExternalAccessible := 'False'; ExternalVisible := 'False'; ExternalWritable := 'False'} : Array[0..0] of "LBC_typeSinaSpeedInterface";
      twoWayActuator { ExternalAccessible := 'False'; ExternalVisible := 'False'; ExternalWritable := 'False'} : Array[0..1] of "LBC_typeTwoWayActuatorInterface";
   END_VAR
BEGIN
   manualOperationEm.equipmentModuleNum := 1040;
END_DATA_BLOCK

DATA_BLOCK "ManualOperationControl_U1Em4"   // DB161
// stored: MemoryReserve 100
   VAR
      manualOperationEm { ExternalAccessible := 'False'; ExternalVisible := 'False'; ExternalWritable := 'False'} : "LAF_typeManEm";
      manualOperationEmArea { ExternalAccessible := 'False'; ExternalVisible := 'False'; ExternalWritable := 'False'} : Array[1..2] of "LAF_typeManOperationArea";
      manualOperationCms { ExternalAccessible := 'False'; ExternalVisible := 'False'; ExternalWritable := 'False'} : Array[1..45] of "LAF_typeManOperation";
      axis { ExternalAccessible := 'False'; ExternalVisible := 'False'; ExternalWritable := 'False'} : Array[0..3] of "LBC_typeAxisControlInterface";
      axis64Pos { ExternalAccessible := 'False'; ExternalVisible := 'False'; ExternalWritable := 'False'} : Array[0..1] of "LBC_typeAxis64PosInterface";
      softCam { ExternalAccessible := 'False'; ExternalVisible := 'False'; ExternalWritable := 'False'} : Array[0..1] of "LER_typeSoftCamRelation";
      sina { ExternalAccessible := 'False'; ExternalVisible := 'False'; ExternalWritable := 'False'} : Array[0..0] of "LBC_typeSinaSpeedInterface";
      twoWayActuator { ExternalAccessible := 'False'; ExternalVisible := 'False'; ExternalWritable := 'False'} : Array[0..1] of "LBC_typeTwoWayActuatorInterface";
   END_VAR
BEGIN
   manualOperationEm.equipmentModuleNum := 1050;
END_DATA_BLOCK

DATA_BLOCK "ManualOperationControl_U1Em5"   // DB157
// stored: MemoryReserve 100
   VAR
      manualOperationEm { ExternalAccessible := 'False'; ExternalVisible := 'False'; ExternalWritable := 'False'} : "LAF_typeManEm";
      manualOperationEmArea { ExternalAccessible := 'False'; ExternalVisible := 'False'; ExternalWritable := 'False'} : Array[1..2] of "LAF_typeManOperationArea";
      manualOperationCms { ExternalAccessible := 'False'; ExternalVisible := 'False'; ExternalWritable := 'False'} : Array[1..45] of "LAF_typeManOperation";
      axis { ExternalAccessible := 'False'; ExternalVisible := 'False'; ExternalWritable := 'False'} : Array[0..0] of "LBC_typeAxisControlInterface";
      axis64Pos { ExternalAccessible := 'False'; ExternalVisible := 'False'; ExternalWritable := 'False'} : Array[0..2] of "LBC_typeAxis64PosInterface";
      softCam { ExternalAccessible := 'False'; ExternalVisible := 'False'; ExternalWritable := 'False'} : Array[0..2] of "LER_typeSoftCamRelation";
      sina { ExternalAccessible := 'False'; ExternalVisible := 'False'; ExternalWritable := 'False'} : Array[0..0] of "LBC_typeSinaSpeedInterface";
      twoWayActuator { ExternalAccessible := 'False'; ExternalVisible := 'False'; ExternalWritable := 'False'} : Array[0..6] of "LBC_typeTwoWayActuatorInterface";
   END_VAR
BEGIN
   manualOperationEm.equipmentModuleNum := 1060;
END_DATA_BLOCK

DATA_BLOCK "ManualOperationControl_U1Em6"   // DB159
// stored: MemoryReserve 100
   VAR
      manualOperationEm { ExternalAccessible := 'False'; ExternalVisible := 'False'; ExternalWritable := 'False'} : "LAF_typeManEm";
      manualOperationEmArea { ExternalAccessible := 'False'; ExternalVisible := 'False'; ExternalWritable := 'False'} : Array[1..2] of "LAF_typeManOperationArea";
      manualOperationCms { ExternalAccessible := 'False'; ExternalVisible := 'False'; ExternalWritable := 'False'} : Array[1..45] of "LAF_typeManOperation";
      axis { ExternalAccessible := 'False'; ExternalVisible := 'False'; ExternalWritable := 'False'} : Array[0..0] of "LBC_typeAxisControlInterface";
      axis64Pos { ExternalAccessible := 'False'; ExternalVisible := 'False'; ExternalWritable := 'False'} : Array[0..1] of "LBC_typeAxis64PosInterface";
      softCam { ExternalAccessible := 'False'; ExternalVisible := 'False'; ExternalWritable := 'False'} : Array[0..1] of "LER_typeSoftCamRelation";
      sina { ExternalAccessible := 'False'; ExternalVisible := 'False'; ExternalWritable := 'False'} : Array[0..0] of "LBC_typeSinaSpeedInterface";
      twoWayActuator { ExternalAccessible := 'False'; ExternalVisible := 'False'; ExternalWritable := 'False'} : Array[0..1] of "LBC_typeTwoWayActuatorInterface";
   END_VAR
BEGIN
   manualOperationEm.equipmentModuleNum := 1070;
END_DATA_BLOCK

DATA_BLOCK "ManualOperationControl_U1Em7"   // DB162
// stored: MemoryReserve 100
   VAR
      manualOperationEm { ExternalAccessible := 'False'; ExternalVisible := 'False'; ExternalWritable := 'False'} : "LAF_typeManEm";
      manualOperationEmArea { ExternalAccessible := 'False'; ExternalVisible := 'False'; ExternalWritable := 'False'} : Array[1..2] of "LAF_typeManOperationArea";
      manualOperationCms { ExternalAccessible := 'False'; ExternalVisible := 'False'; ExternalWritable := 'False'} : Array[1..45] of "LAF_typeManOperation";
      axis { ExternalAccessible := 'False'; ExternalVisible := 'False'; ExternalWritable := 'False'} : Array[0..6] of "LBC_typeAxisControlInterface";
      axis64Pos { ExternalAccessible := 'False'; ExternalVisible := 'False'; ExternalWritable := 'False'} : Array[0..0] of "LBC_typeAxis64PosInterface";
      softCam { ExternalAccessible := 'False'; ExternalVisible := 'False'; ExternalWritable := 'False'} : Array[0..0] of "LER_typeSoftCamRelation";
      sina { ExternalAccessible := 'False'; ExternalVisible := 'False'; ExternalWritable := 'False'} : Array[0..3] of "LBC_typeSinaSpeedInterface";
      twoWayActuator { ExternalAccessible := 'False'; ExternalVisible := 'False'; ExternalWritable := 'False'} : Array[0..1] of "LBC_typeTwoWayActuatorInterface";
   END_VAR
BEGIN
   manualOperationEm.equipmentModuleNum := 1080;
END_DATA_BLOCK

DATA_BLOCK "DriveDiagConfig"   // DB18
TITLE = DriveDiagConfig
AUTHOR : Siemens Digital Industries
FAMILY : LAF
NAME : LAF_DriveDiagConfigData
VERSION : 1.1
// Configuration data array for drive diagnostic
// stored: MemoryReserve 100
   VAR
      driveObjects : Array[0.."LAF_DRV_DIAG_NO_DO"] of "LAF_typeDriveDiagConfig";
   END_VAR
BEGIN
END_DATA_BLOCK

DATA_BLOCK "DriveDiagInterfaceHmi"   // DB46
TITLE = DriveDiagInterfaceHmi
AUTHOR : Siemens Digital Industries
FAMILY : LAF
NAME : LAF_DriveDiagInterfaceHmi
VERSION : 1.1
// HMI interface for drive diagnostic
// stored: MemoryReserve 100
   VAR
      diagStatus : "LAF_typeDriveDiagInterfaceHmi";
   END_VAR
BEGIN
END_DATA_BLOCK

DATA_BLOCK "IdentData"   // DB221
TITLE = Schnittstelle Read/Write Daten / Interface read/write data
AUTHOR : SICAR
FAMILY : Ident
VERSION : 1.0
// Ident Daten / Ident data
// stored: MemoryReserve 100
   VAR
      rfReader { ExternalAccessible := 'False'; ExternalVisible := 'False'; ExternalWritable := 'False'} : Array[0.."NO_OF_RF_IDENT_DEVICES"] of "LSicar_typeIdentReadWriteDat";   // Reader
   END_VAR
BEGIN
END_DATA_BLOCK

DATA_BLOCK "InterfaceSignals"   // DB182
// stored: MemoryReserve 100
   VAR
      HMI_Interface_Mode : Bool;
      "Button Value" : Array[0..16] of "LER_SignalsInput";
   END_VAR
BEGIN
END_DATA_BLOCK

DATA_BLOCK "SafetyDoorInterface"   // DB188
// stored: MemoryReserve 100
   VAR
      "FDoorEC.LH" { ExternalWritable := 'False'} : "LER_typefDoorInterface";
      "FDoorEC.RH" { ExternalWritable := 'False'} : "LER_typefDoorInterface";
      "FDoorEC.Top" { ExternalWritable := 'False'} : "LER_typefDoorInterface";
      FDoorCutter : "LER_typefDoorInterface";
      FDoorMagazine : "LER_typefDoorInterface";
      FDoorConveyor : "LER_typefDoorInterface";
      FDoorCentralAisle : "LER_typefDoorInterface";
   END_VAR
BEGIN
   "FDoorEC.LH".configuration.referenceDesignator := WSTRING#'LH';
   "FDoorEC.RH".configuration.referenceDesignator := WSTRING#'RH';
   "FDoorEC.Top".configuration.referenceDesignator := WSTRING#'Main';
   FDoorCutter.configuration.referenceDesignator := WSTRING#'Cutter';
   FDoorMagazine.configuration.referenceDesignator := WSTRING#'Magazine';
   FDoorConveyor.configuration.referenceDesignator := WSTRING#'C/V';
   FDoorCentralAisle.configuration.referenceDesignator := WSTRING#'Central';
END_DATA_BLOCK

DATA_BLOCK "DI1"   // DB279
// stored: MemoryReserve 100
   VAR
      "MOTOR POWER TRIPPED E202CB" : Bool;
      "REELCUT CONVEYOR RING BLOW POWER TRIPPED" : Bool;
      "STACKING-1 CONVEYOR RING BLOW POWER TRIPPED E214CB" : Bool;
      "STACKING-2 CONVEYOR RING BLOW POWER TRIPPED E220CB" : Bool;
      SPARE1 : Bool;
      "E6404PWS CONTROLLER POWER SMPS AC POWER TRIPPED E320CB" : Bool;
      "E6704PWS CONTROLLER POWER SMPS AC POWER TRIPPED E326CB" : Bool;
      "E6804PWS SAFETY POWER SMPS AC POWER TRIPPED E332CB" : Bool;
      SPARE2 : Bool;
      "POWER METER POWER TRIPPED E720CB" : Bool;
      "POWER METER CONTROL POWER TRIPPED E726CB" : Bool;
      SPARE3 : Bool;
      "PROCESSOR POWER ON TRIPPED E4116CB" : Bool;
      "PROGRAMMING POWER OUTLET TRIPPED E4156CB" : Bool;
      SPARE4 : Bool;
      "PANEL LED POWER TRIPPED E4304CB" : Bool;
      SPARE5 : Bool;
      "PLC POWER SMPS DC OK E4404PWS" : Bool;
      "CONTROL LEVEL HUB POWER TRIPPED E4420CB" : Bool;
      "MAIN HMI POWER TRIPPED E4426CB" : Bool;
      "PORTABLE HMI POWER TRIPPED E4432CB" : Bool;
      "PORTABLE HMI POWER TRIPPED E4456CB" : Bool;
      SPARE6 : Bool;
      SPARE7 : Bool;
      "120VAC CONTROL POWER TR PRIMARY TRIPPED E5100CB" : Bool;
      "120VAC CONTROL POWER TR SECONDARY TRIPPED E5110CB" : Bool;
      "CONTROL POWER ON TRIPPED E5116CB" : Bool;
      "VISION MONITOR POWER STRIP OUTLET POWER TRIPPED E5160CB" : Bool;
      "MCU & RFD HANDY POWER STRIP OUTLET POWER TRIPPED E5166CB" : Bool;
      "VISION LIGHT CONTROLLER POWER STRIP OUTLET POWER TRIPPED E5172CB" : Bool;
      SPARE8 : Bool;
      "FFU POWER-1 POWER TRIPPED E3222CB" : Bool;
   END_VAR
BEGIN
END_DATA_BLOCK

DATA_BLOCK "DI2"   // DB290
// stored: MemoryReserve 100
   VAR
      SPARE1 : Bool;
      "CONTROL POWER SMPS DC OK E6104PWS" : Bool;
      "ET200MP I/O OUTPUT POWER TRIPPED E6154CB" : Bool;
      "JUNCTION BOX CONTROL POWER TRIPPED E6180CB" : Bool;
      "CLASS 2 SMPS POWER TRIPPED E6204CB" : Bool;
      "CLASS 2 SMPS MONITORING E6206PWS" : Bool;
      "ET200ECO PN-1 POWER TRIPPED E6220CB" : Bool;
      "ET200ECO PN-2 POWER TRIPPED E6224CB" : Bool;
      "ET200ECO PN-3 POWER TRIPPED E6228CB" : Bool;
      SPARE2 : Bool;
      "PANEL FAN POWER TRIPPED E6304CB" : Bool;
      SPARE3 : Bool;
      "CONTROLLER POWER SMPS DC OK E6404PWS" : Bool;
      "CONTROLLER DC POWER TRIPPED E6406CB" : Bool;
      "SERVO CONTROL POWER TRIPPED E6416CB" : Bool;
      "MANIFOLD-1 CONTROL POWER TRIPPED E6422CB" : Bool;
      SPARE4 : Bool;
      "RFID POWER TRIPPED E6456CB" : Bool;
      "QR READER POWER TRIPPED E6462CB" : Bool;
      "QR READER POWER TRIPPED E6468CB" : Bool;
      SPARE5 : Bool;
      SPARE6 : Bool;
      "CONTROLLER POWER SMPS DC OK E6704PWS" : Bool;
      "CONTROLLER DC POWER TRIPPED E6706CB" : Bool;
      "HANDY QR READER POWER TRIPPED E6716CB" : Bool;
      "VISION CONTROLLER POWER TRIPPED E6722CB" : Bool;
      "LINE LASER MODULE-1 POWER TRIPPED E6728CB" : Bool;
      "LINE LASER MODULE-2 POWER TRIPPED E6734CB" : Bool;
      "EPC CONTROLLER-1 POWER TRIPPED E6756CB" : Bool;
      "EPC CONTROLLER-2 POWER TRIPPED E6762CB" : Bool;
      "EPC CONTROLLER-3 POWER TRIPPED E6768CB" : Bool;
      "DRIVE-CLIQ HUB POWER TRIPPED E6774CB" : Bool;
   END_VAR
BEGIN
END_DATA_BLOCK

DATA_BLOCK "DI3"   // DB280
// stored: MemoryReserve 100
   VAR
      "EQUIPMENT LED POWER TRIPPED E6780CB" : Bool;
      "MOTOR POWER MC COIL POWER TRIPPED E6786CB" : Bool;
      "SAFETY POWER SMPS DC OK E6804PWS" : Bool;
      "SAFETY DC POWER TRIPPED E6808CB" : Bool;
      "ET200SP I/O SAFETY POWER TRIPPED E6816CB" : Bool;
      "JUNCTION BOX CONTROL POWER TRIPPED E6836CB" : Bool;
      "ET200ECO PN-SAFETY-1 POWER TRIPPED E6856CB" : Bool;
      SPARE1 : Bool;
      SPARE2 : Bool;
      SPARE3 : Bool;
      SPARE4 : Bool;
      SPARE5 : Bool;
      SPARE6 : Bool;
      SPARE7 : Bool;
      SPARE8 : Bool;
      SPARE9 : Bool;
      SPARE10 : Bool;
      SPARE11 : Bool;
      SPARE12 : Bool;
      SPARE13 : Bool;
      SPARE14 : Bool;
      SPARE15 : Bool;
      SPARE16 : Bool;
      SPARE17 : Bool;
      SPARE18 : Bool;
      SPARE19 : Bool;
      SPARE20 : Bool;
      SPARE21 : Bool;
      SPARE22 : Bool;
      SPARE23 : Bool;
      SPARE24 : Bool;
      SPARE25 : Bool;
   END_VAR
BEGIN
END_DATA_BLOCK

DATA_BLOCK "DQ1"   // DB289
// stored: MemoryReserve 100
   VAR
      "EQUIPMENT LED LAMP RELAY ON" : Bool;
      SPARE1 : Bool;
      SPARE2 : Bool;
      "CLASS2 SMPS ALARM RESET" : Bool;
      SPARE3 : Bool;
      SPARE4 : Bool;
      SPARE5 : Bool;
      SPARE6 : Bool;
      SPARE7 : Bool;
      SPARE8 : Bool;
      SPARE9 : Bool;
      SPARE10 : Bool;
      SPARE11 : Bool;
      SPARE12 : Bool;
      SPARE13 : Bool;
      SPARE14 : Bool;
      SPARE15 : Bool;
      SPARE16 : Bool;
      SPARE17 : Bool;
      SPARE18 : Bool;
      SPARE19 : Bool;
      SPARE20 : Bool;
      SPARE21 : Bool;
      SPARE22 : Bool;
      SPARE23 : Bool;
      SPARE24 : Bool;
      SPARE25 : Bool;
      SPARE26 : Bool;
      SPARE27 : Bool;
      SPARE28 : Bool;
      SPARE29 : Bool;
      SPARE30 : Bool;
   END_VAR
BEGIN
END_DATA_BLOCK

DATA_BLOCK "FDI1"   // DB292
// stored: MemoryReserve 100
   VAR
      "MANIFOLD-1 SOL POWER MC FEEDBACK" : Bool;
      "MANIFOLD-2 SOL POWER MC FEEDBACK" : Bool;
      SPARE1 : Bool;
      SPARE2 : Bool;
      "FFU POWER MC 1 FEEDBACK" : Bool;
      "FFU POWER MC 2 FEEDBACK" : Bool;
      SPARE3 : Bool;
      SPARE4 : Bool;
   END_VAR
BEGIN
END_DATA_BLOCK

DATA_BLOCK "FDQ1"   // DB291
// stored: MemoryReserve 100
   VAR
      "MANIFOLD-1 SOL POWER MC ON" : Bool;
      SPARE1 : Bool;
      SPARE2 : Bool;
      SPARE3 : Bool;
      "FFU POWER MC ON 1" : Bool;
      "FFU POWER MC ON 2" : Bool;
      SPARE4 : Bool;
      SPARE5 : Bool;
   END_VAR
BEGIN
END_DATA_BLOCK

DATA_BLOCK "BK01"   // DB222
// stored: MemoryReserve 100
   VAR
      "X10-1 LEFT UNWINDER EXPEL BACKWARD" : Bool;
      "X11-1 RIGHT UNWINDER EXPEL BACKWARD" : Bool;
      "X12-1 UW SUPPORT UNIT TRANSFER BACKWARD" : Bool;
      "X13-1 ELECTRODE SHAFT SUPPORTER DOWN" : Bool;
      "X14-1 LEFT TENSION CHECK SENSOR" : Bool;
      "X15-1 ELECTRODE FIX LEFT TOP PRESSURE SWITCH" : Bool;
      "X16-1 SPARE" : Bool;
      "X17-1 SPARE" : Bool;
      "X10-2 LEFT UNWINDER EXPEL FORWARD" : Bool;
      "X11-2 RIGHT UNWINDER EXPEL FORWARD" : Bool;
      "X12-2 UW SUPPORT UNIT TRANSFER FORWARD" : Bool;
      "X13-2 ELECTRODE SHAFT SUPPORTER UP" : Bool;
      "X14-2 RIGHT TENSION CHECK SENSOR" : Bool;
      "X15-2 ELECTRODE FIX LEFT BTM PRESSURE SWITCH" : Bool;
      "X16-2 SPARE" : Bool;
      "X17-2 SPARE" : Bool;
   END_VAR
BEGIN
END_DATA_BLOCK

DATA_BLOCK "BK02"   // DB191
// stored: MemoryReserve 100
   VAR
      "X10-1 ELECTRODE FIX RIGHT TOP BACKWARD" : Bool;
      "X10-2 ELECTRODE FIX RIGHT TOP FORWARD" : Bool;
      "X12-1 ELECTRODE FIX RIGHT BTM BACKWARD" : Bool;
      "X12-2 ELECTRODE FIX RIGHT BTM FORWARD" : Bool;
      "X14-1 ELECTRODE FIX RIGHT TOP PRESSURE SWITCH" : Bool;
      "X14-2 ELECTRODE FIX RIGHT BTM PRESSURE SWITCH" : Bool;
      "X16-1 ELECTRODE CUTTER BACKWARD" : Bool;
      "X16-2 ELECTRODE CUTTER FORWARD" : Bool;
   END_VAR
BEGIN
END_DATA_BLOCK

DATA_BLOCK "BK03"   // DB192
// stored: MemoryReserve 100
   VAR
      "X10-1 ELECTRODE FIX LEFT TOP BACKWARD" : Bool;
      "X11-1 UNWINDER STOPPER BACKWARD" : Bool;
      "X12-1 ELECTRODE FIX LEFT BTM BACKWARD" : Bool;
      "X13-1 DIGITAL PRESSURE SWITCH OUT1" : Bool;
      "X14-1 ELECTRODE FIX LEFT TOP UP" : Bool;
      "X15-1 FRAME COVER BACKWARD" : Bool;
      "X16-1 ELECTRODE FIX LEFT BTM DOWN" : Bool;
      "X17-1 SPARE" : Bool;
      "X10-2 ELECTRODE FIX LEFT TOP FORWARD" : Bool;
      "X11-2 UNWINDER STOPPER FORWARD" : Bool;
      "X12-2 ELECTRODE FIX LEFT BTM FORWARD" : Bool;
      "X13-2 DIGITAL PRESSURE SWITCH OUT2" : Bool;
      "X14-2 ELECTRODE FIX LEFT TOP DOWN" : Bool;
      "X15-2 FRAME COVER FORWARD" : Bool;
      "X16-2 ELECTRODE FIX LEFT BTM UP" : Bool;
      "X17-2 SPARE" : Bool;
   END_VAR
BEGIN
END_DATA_BLOCK

DATA_BLOCK "BK04"   // DB193
// stored: MemoryReserve 100
   VAR
      "X10-1 SPLICING L-MODULE MOVER BACKWARD" : Bool;
      "X11-1 SPLICING R-MODULE MOVER BACKWARD" : Bool;
      "X12-1 ELECTRODE L-HOLDER MOVER FORWARD" : Bool;
      "X13-1 ELECTRODE R-HOLDER MOVER FORWARD" : Bool;
      "X14-1 TAPE LOADING TURN HOMING" : Bool;
      "X15-1 TAPE ATTACH UNIT BACKWARD" : Bool;
      "X16-1 TAPING VACUUM PRESSURE SWITCH" : Bool;
      "X17-1 SPARE" : Bool;
      "X10-2 SPLICING L-MODULE MOVER FORWARD" : Bool;
      "X11-2 SPLICING R-MODULE MOVER FORWARD" : Bool;
      "X12-2 ELECTRODE L-HOLDER MOVER BACKWARD" : Bool;
      "X13-2 ELECTRODE R-HOLDER MOVER BACKWARD" : Bool;
      "X14-2 TAPE LOADING TURN ROTATE" : Bool;
      "X15-2 TAPE ATTACH UNIT FORWARD" : Bool;
      "X16-2 SPARE" : Bool;
      "X17-2 SPARE" : Bool;
   END_VAR
BEGIN
END_DATA_BLOCK

DATA_BLOCK "BK05"   // DB194
// stored: MemoryReserve 100
   VAR
      "X10-1 SPARE" : Bool;
      "X11-1 SPARE" : Bool;
      "X12-1 COMPENSATOR LIMIT SENSOR(-)" : Bool;
      "X13-1 COMPENSATOR LIMIT SENSOR(+)" : Bool;
      "X14-1 FEEDER CYLINDER UP" : Bool;
      "X15-1 VISION PUSHER SUPPORT UP" : Bool;
      "X16-1 ELECTRODE NG BOX LOCK CYLINDER DOWN" : Bool;
      "X17-1 UNWINDER DANCER SAFETY PIN IDLE POSITION" : Bool;
      "X10-2 SPARE" : Bool;
      "X11-2 SPARE" : Bool;
      "X12-2 COMPENSATOR HOMING SENSOR" : Bool;
      "X13-2 COMPENSATOR SAFETY PIN IDLE POSITION" : Bool;
      "X14-2 FEEDER CYLINDER DOWN" : Bool;
      "X15-2 VISION PUSHER SUPPORT DOWN" : Bool;
      "X16-2 ELECTRODE NG BOX LOCK CYLINDER UP" : Bool;
      "X17-2 SPARE" : Bool;
   END_VAR
BEGIN
END_DATA_BLOCK

DATA_BLOCK "BK06"   // DB201
// stored: MemoryReserve 100
   VAR
      "X10-1 NG & MANUAL INPUT CYLINDER UP" : Bool;
      "X11-1 MAGAZINE LOCK CYLINDER DOWN" : Bool;
      "X12-1 NG & MANUAL INPUT PAD VACUUM PRESSURE SWITCH" : Bool;
      "X13-1 NG & MANUAL INPUT LIMIT SENSOR(-)" : Bool;
      "X14-1 NG & MANUAL INPUT LIMIT SENSOR(+)" : Bool;
      "X15-1 NG & MANUAL INPUT MAGAZINE LIMIT SENSOR(-)" : Bool;
      "X16-1 NG & MANUAL INPUT MAGAZINE LIMIT SENSOR(+)" : Bool;
      "X17-1 NG & MANUAL INPUT MAGAZINE ELECTRODE DETECTION SENSOR" : Bool;
      "X10-2 NG & MANUAL INPUT CYLINDER DOWN" : Bool;
      "X11-2 MAGAZINE LOCK CYLINDER UP" : Bool;
      "X12-2 NG & MANUAL INPUT VIBRATOR VACUUM PRESSURE SWITCH" : Bool;
      "X13-2 NG & MANUAL INPUT HOMING SENSOR" : Bool;
      "X14-2 NG & MANUAL INPUT ELECTRODE DETECTION SENSOR" : Bool;
      "X15-2 NG & MANUAL INPUT MAGAZINE HOMING SENSOR" : Bool;
      "X16-2 SPARE" : Bool;
      "X17-2 NG & MANUAL INPUT MAGAZINE DETECTION SENSOR" : Bool;
   END_VAR
BEGIN
END_DATA_BLOCK

DATA_BLOCK "BK07"   // DB202
// stored: MemoryReserve 100
   VAR
      "X10-1 POSITION MOVING LIMIT SENSOR(-)" : Bool;
      "X11-1 POSITION MOVING LIMIT SENSOR(+)" : Bool;
      "X12-1 VISION HOMING SENSOR" : Bool;
      "X13-1 ELECTRODE NG KICKER HOMING SENSOR" : Bool;
      "X14-1 ELECTRODE NG BOX FULL SENSOR" : Bool;
      "X15-1 ELECTRODE NG BOX DETECT SENSOR" : Bool;
      "X16-1 NG & MANUAL INPUT MAGAZINE FULL SENSOR" : Bool;
      "X17-1 MAGAZINE Z-AXIS SAFETY PIN POSITION SENSOR" : Bool;
      "X10-2 POSITION MOVING HOMING SENSOR" : Bool;
      "X11-2 CUTTER HOMING SENSOR" : Bool;
      "X12-2 SPARE" : Bool;
      "X13-2 ELECTRODE PASS KICKER HOMING SENSOR" : Bool;
      "X14-2 SPARE" : Bool;
      "X15-2 SPARE" : Bool;
      "X16-2 SPARE" : Bool;
      "X17-2 SPARE" : Bool;
   END_VAR
BEGIN
END_DATA_BLOCK

DATA_BLOCK "BK08"   // DB203
// stored: MemoryReserve 100
   VAR
      "X10-1 UW ELECTRODE FIX LEFT TOP V/C ON" : Bool;
      "X10-2 UW ELECTRODE FIX LEFT TOP V/C OFF" : Bool;
      "X12-1 UW ELECTRODE FIX LEFT BTM V/C ON" : Bool;
      "X12-2 UW ELECTRODE FIX LEFT BTM V/C OFF" : Bool;
      "X14-1 UW ELECTRODE FIX RIGHT TOP V/C ON" : Bool;
      "X14-2 UW ELECTRODE FIX RIGHT TOP V/C OFF" : Bool;
      "X16-1 UW ELECTRODE FIX RIGHT BTM V/C ON" : Bool;
      "X16-2 UW ELECTRODE FIX RIGHT BTM V/C OFF" : Bool;
   END_VAR
BEGIN
END_DATA_BLOCK

DATA_BLOCK "BK09"   // DB204
// stored: MemoryReserve 100
   VAR
      "X10-1 NG & MANUAL INPUT VIBRATOR-1 ON" : Bool;
      "X10-2 NG & MANUAL INPUT VIBRATOR-1 OFF" : Bool;
      "X12-1 NG & MANUAL INPUT PAD VACUUM ON" : Bool;
      "X12-2 NG & MANUAL INPUT PAD VACUUM OFF" : Bool;
      "X14-1 NG & MANUAL INPUT VIBRATOR VACUUM ON" : Bool;
      "X14-2 NG & MANUAL INPUT VIBRATOR VACUUM OFF" : Bool;
      "X16-1 NG & MANUAL INPUT VIBRATOR-2 ON" : Bool;
      "X16-2 NG & MANUAL INPUT VIBRATOR-2 OFF" : Bool;
   END_VAR
BEGIN
END_DATA_BLOCK

DATA_BLOCK "BK10"   // DB205
// stored: MemoryReserve 100
   VAR
      "X10-1 UW TAPE ATTACH V/C ON" : Bool;
      "X10-2 UW TAPE ATTACH V/C OFF" : Bool;
      "X12-1 CART DETECT CHECK LAMP" : Bool;
      "X12-2 SPARE" : Bool;
      "X14-1 SPARE" : Bool;
      "X14-2 SPARE" : Bool;
      "X16-1 SPARE" : Bool;
      "X16-2 SPARE" : Bool;
   END_VAR
BEGIN
END_DATA_BLOCK

DATA_BLOCK "ET200SP_201"   // DB227
// stored: MemoryReserve 100
   VAR
      "SP201.00 AUTO INITIATE PBL (GREEN)" : Bool;
      "SP201.01 STOP PBL (RED)" : Bool;
      SPARE1 : Bool;
      SPARE2 : Bool;
      SPARE3 : Bool;
      SPARE4 : Bool;
      SPARE5 : Bool;
      SPARE6 : Bool;
      "SP201.08 MAIN HMI POWER TRIPPED E110CB" : Bool;
      SPARE7 : Bool;
      SPARE8 : Bool;
      SPARE9 : Bool;
      SPARE10 : Bool;
      SPARE11 : Bool;
      SPARE12 : Bool;
      SPARE13 : Bool;
   END_VAR
BEGIN
END_DATA_BLOCK

DATA_BLOCK "ET200SP_202"   // DB273
// stored: MemoryReserve 100
   VAR
      "SP202.00 AUTO INITIATE PBL LAMP ON (GREEN)" : Bool;
      "SP202.01 STOP PBL LAMP ON (RED)" : Bool;
      SPARE1 : Bool;
      "SP202.03 ENABLE PBL LAMP ON (BLACK)" : Bool;
      "SP202.04 SAFETY RESET PBL LAMP ON (BLUE)" : Bool;
      SPARE2 : Bool;
      SPARE3 : Bool;
      SPARE4 : Bool;
      "SP202.08 TOWER LAMP 1 ON (RED)" : Bool;
      "SP202.09 TOWER LAMP 2 ON (AMBER)" : Bool;
      "SP202.10 TOWER LAMP 3 ON (GREEN)" : Bool;
      "SP202.11 TOWER LAMP 4 ON (WHITE)" : Bool;
      "SP202.12 TOWER LAMP 5 ON (BLUE)" : Bool;
      "SP202.13 TOWER LAMP 6 ON (BUZZER)" : Bool;
      SPARE5 : Bool;
      SPARE6 : Bool;
   END_VAR
BEGIN
END_DATA_BLOCK

DATA_BLOCK "ET200SP_203"   // DB272
// stored: MemoryReserve 100
   VAR
      "SP203.00 Main OP: mode select, Auto" : Bool;
      "SP203.01 Main OP: home (GREEN)" : Bool;
      "SP203.02 Main OP: safety reset (BLUE)" : Bool;
      "SP203.03 Main OP: SCS mode select, Auto" : Bool;
      "SP203.04 Main OP: mode select, Manual" : Bool;
      "SP203.05 Main OP: enable" : Bool;
      "SP203.06 Main OP: SCS mode select, Setup" : Bool;
      "SP203.07 Main OP: SCS mode select, Disable" : Bool;
   END_VAR
BEGIN
END_DATA_BLOCK

DATA_BLOCK "ET200SP_204"   // DB296
// stored: MemoryReserve 100
   VAR
      "SP204.00 Main OP: Emergency stop" : Bool;
      SPARE1 : Bool;
      SPARE2 : Bool;
      SPARE3 : Bool;
      RESERVED : Bool;
      SPARE4 : Bool;
      SPARE5 : Bool;
      SPARE6 : Bool;
   END_VAR
BEGIN
END_DATA_BLOCK

DATA_BLOCK "ET200SP_205"   // DB274
// stored: MemoryReserve 100
   VAR
      "SP205.00 Main OP: pendant required on, yellow" : Bool;
      SPARE1 : Bool;
      "SP205.02 Main OP: home on, green" : Bool;
      SPARE2 : Bool;
      SPARE3 : Bool;
      SPARE4 : Bool;
      SPARE5 : Bool;
      "SP205.07 Main OP: SCS Disable mode selected, green" : Bool;
   END_VAR
BEGIN
END_DATA_BLOCK

DATA_BLOCK "ET500SP_501"   // DB228
// stored: MemoryReserve 100
   VAR
      "SP501.00 CONTROL DC POWER TRIPPED E156CB" : Bool;
      "SP501.01 SAFETY DC POWER TRIPPED E218CB" : Bool;
      SPARE1 : Bool;
      SPARE2 : Bool;
      "SP501.04 Vision STO" : Bool;
      "SP501.05 Vision Judgment" : Bool;
      SPARE3 : Bool;
      SPARE4 : Bool;
      SPARE5 : Bool;
      SPARE6 : Bool;
      SPARE7 : Bool;
      SPARE8 : Bool;
      SPARE9 : Bool;
      SPARE10 : Bool;
      SPARE11 : Bool;
      SPARE12 : Bool;
   END_VAR
BEGIN
END_DATA_BLOCK

DATA_BLOCK "ET500SP_502"   // DB231
// stored: MemoryReserve 100
   VAR
      SPARE1 : Bool;
      SPARE2 : Bool;
      SPARE3 : Bool;
      SPARE4 : Bool;
      SPARE5 : Bool;
      SPARE6 : Bool;
      SPARE7 : Bool;
      SPARE8 : Bool;
      SPARE9 : Bool;
      SPARE10 : Bool;
      SPARE11 : Bool;
      SPARE12 : Bool;
      SPARE13 : Bool;
      SPARE14 : Bool;
      SPARE15 : Bool;
      SPARE16 : Bool;
   END_VAR
BEGIN
END_DATA_BLOCK

DATA_BLOCK "ET500SP_503"   // DB249
// stored: MemoryReserve 100
   VAR
      "SP503.00 LEFT UNWINDER RADIUS MEASURE" : LReal;
      "SP503.01 RIGHT UNWINDER RADIUS MEASURE" : LReal;
      "SP503.02 UNWINDER LOADCELL" : LReal;
      "SP503.03 CUTTER EPC SENSOR" : LReal;
   END_VAR
BEGIN
END_DATA_BLOCK

DATA_BLOCK "ET500SP_504"   // DB229
// stored: MemoryReserve 100
   VAR
      "SP504.00 UNWINDER DANCER ENCODER" : Int;
      SPARE1 : Int;
      SPARE2 : Int;
      SPARE3 : Int;
   END_VAR
BEGIN
END_DATA_BLOCK

DATA_BLOCK "ET500SP_505"   // DB235
// stored: MemoryReserve 100
   VAR
      "SP505.00 UNWINDER DANCER ELECTRO-PNEUMATIC REGULATOR" : LReal;
      SPARE1 : LReal;
      SPARE2 : LReal;
      SPARE3 : LReal;
   END_VAR
BEGIN
END_DATA_BLOCK

DATA_BLOCK "ET500SP_506"   // DB234
// stored: MemoryReserve 100
   VAR
      "SP506.00 Tab Sensor" : Bool;
      "SP506.01 Tape Sensor" : Bool;
      "SP506.02 VISION TRIGGER SENSOR" : Bool;
      "SP506.03 ELECTRODE PASS KICKER DETECT SENSOR" : Bool;
      "SP506.04 OutputCam_FeedingRollAxisB" : Bool;
      "SP506.05 OutputCam_ElectrodeCutterAxisZ" : Bool;
      "SP506.06 VISION CONTROLLER TRIGGER" : Bool;
      "SP506.07 OutputCam_NgKickerAxisZ" : Bool;
      SPARE1 : Bool;
   END_VAR
BEGIN
END_DATA_BLOCK

DATA_BLOCK "ET500SP_507"   // DB236
// stored: MemoryReserve 100
   VAR
      "SP507.00 ELECTRODE NG KICKER DETECT SENSOR" : Bool;
      "SP507.01 ELECTRODE DETECT COLOR SENSOR #1" : Bool;
      "SP507.02 ELECTRODE DETECT COLOR SENSOR #2" : Bool;
      SPARE1 : Bool;
      "SP507.04 OutputCam_PassKickerAxisZ" : Bool;
      SPARE2 : Bool;
      SPARE3 : Bool;
      SPARE4 : Bool;
      SPARE5 : Bool;
   END_VAR
BEGIN
END_DATA_BLOCK

DATA_BLOCK "ET500SP_508"   // DB230
// stored: MemoryReserve 100
   VAR
      "SP508.00 PHMI-1 EMERGENCY STOP" : Bool;
      "SP508.01 PHMI-1 ENABLE SWITCH" : Bool;
      "SP508.02 PHMI-2 EMERGENCY STOP" : Bool;
      "SP508.03 PHMI-2 ENABLE SWITCH" : Bool;
      SPARE1 : Bool;
      SPARE2 : Bool;
      SPARE3 : Bool;
      SPARE4 : Bool;
   END_VAR
BEGIN
END_DATA_BLOCK

DATA_BLOCK "ET500SP_509"   // DB233
// stored: MemoryReserve 100
   VAR
      "SP509.00 UNWINDER EPCC01 INTERKOCK" : Bool;
      "SP509.01 UNWINDER EPCC02 INTERLOCK" : Bool;
      "SP509.02 UNWINDER EPCC03 INTERLOCK" : Bool;
      SPARE1 : Bool;
      SPARE2 : Bool;
      SPARE3 : Bool;
      SPARE4 : Bool;
      SPARE5 : Bool;
   END_VAR
BEGIN
END_DATA_BLOCK

DATA_BLOCK "ET500SP_513"   // DB278
// stored: MemoryReserve 100
   VAR
      "SP513.00 LEFT UNWINDER RADIUS SENSOR" : Int;
      "SP513.01 RIGHT UNWINDER RADIUS SENSOR" : Int;
      SPARE1 : Int;
      SPARE2 : Int;
   END_VAR
BEGIN
END_DATA_BLOCK

DATA_BLOCK "PM01"   // DB207
// stored: MemoryReserve 100
   VAR
      "AIRS01 UNWINDER LEFT AIR SHAFT ON" : Bool;
      SPARE_1 : Bool;
      "AIRS02 UNWINDER RIGHT AIR SHAFT ON" : Bool;
      SPARE_2 : Bool;
      SPARE_3 : Bool;
      SPARE_4 : Bool;
      SPARE_5 : Bool;
      SPARE_6 : Bool;
      "C03 UNWINDER SUPPORT UNIT TRANSFER FORWARD" : Bool;
      "C03 UNWINDER SUPPORT UNIT TRANSFER BACKWARD" : Bool;
      "C04 ELECTRODE SHAFT SUPPORTER UP" : Bool;
      "C04 ELECTRODE SHAFT SUPPORTER DOWN" : Bool;
      SPARE_7 : Bool;
      SPARE_8 : Bool;
      SPARE_9 : Bool;
      SPARE_10 : Bool;
   END_VAR
BEGIN
END_DATA_BLOCK

DATA_BLOCK "PM02"   // DB217
// stored: MemoryReserve 100
   VAR
      "C05 UNWINDER SPLICER RIGHT ELECTRODE FIX RIGHT TOP FORWARD" : Bool;
      "C05 UNWINDER SPLICER RIGHT ELECTRODE FIX RIGHT TOP BACKWARD" : Bool;
      "C06 UNWINDER SPLICER RIGHT ELECTRODE FIX RIGHT BTM FORWARD" : Bool;
      "C06 UNWINDER SPLICER RIGHT ELECTRODE FIX RIGHT BTM BACKWARD" : Bool;
      "C07 UNWINDER SPLICER RIGHT CUTTER FORWARD" : Bool;
      "C07 UNWINDER SPLICER RIGHT CUTTER BACKWARD" : Bool;
      "C08 UNWINDER SPLICER LEFT ELECTRODE FIX LEFT TOP FORWARD" : Bool;
      "C08 UNWINDER SPLICER LEFT ELECTRODE FIX LEFT TOP BACKWARD" : Bool;
      "C09 UNWINDER SPLICER LEFT ELECTRODE FIX LEFT BTM FORWARD" : Bool;
      "C09 UNWINDER SPLICER LEFT ELECTRODE FIX LEFT BTM BACKWARD" : Bool;
      "C10 UNWINDER SPLICER LEFT ELECTRODE FIX LEFT TOP DOWN" : Bool;
      "C10 UNWINDER SPLICER LEFT ELECTRODE FIX LEFT TOP UP" : Bool;
      "C11 UNWINDER SPLICER LEFT ELECTRODE FIX LEFT BTM UP" : Bool;
      "C11 UNWINDER SPLICER LEFT ELECTRODE FIX LEFT BTM DOWN" : Bool;
      SPARE_1 : Bool;
      SPARE_2 : Bool;
   END_VAR
BEGIN
END_DATA_BLOCK

DATA_BLOCK "PM03"   // DB219
// stored: MemoryReserve 100
   VAR
      "C12 UNWINDER SPLICER HOLDER SPLICING LEFT MODULE MOVER FORWARD" : Bool;
      "C12 UNWINDER SPLICER HOLDER SPLICING LEFT MODULE MOVER BACKWARD" : Bool;
      "C13 UNWINDER SPLICER HOLDER SPLICING RIGHT MODULE MOVER FORWARD" : Bool;
      "C13 UNWINDER SPLICER HOLDER SPLICING RIGHT MODULE MOVER BACKWARD" : Bool;
      "C14 UNWINDER SPLICER HOLDER ELECTRODE LEFT HOLDER MODULE MOVER FORWARD" : Bool;
      "C14 UNWINDER SPLICER HOLDER ELECTRODE LEFT HOLDER MODULE MOVER BACKWARD" : Bool;
      "C15 UNWINDER SPLICER HOLDER ELECTRODE RIGHT HOLDER MODULE MOVER FORWARD" : Bool;
      "C15 UNWINDER SPLICER HOLDER ELECTRODE RIGHT HOLDER MODULE MOVER BACKWARD" : Bool;
      "C16 UNWINDER SPLICER TAPE LOADING TURN ROTATE" : Bool;
      "C16 UNWINDER SPLICER TAPE LOADING TURN HOME" : Bool;
      "C17 UNWINDER SPLICER TAPE ATTACH UNIT FORWARD" : Bool;
      "C17 UNWINDER SPLICER TAPE ATTACH UNIT BACKWARD" : Bool;
      SPARE_1 : Bool;
      SPARE_2 : Bool;
      SPARE_3 : Bool;
      SPARE_4 : Bool;
   END_VAR
BEGIN
END_DATA_BLOCK

DATA_BLOCK "PM04"   // DB220
// stored: MemoryReserve 100
   VAR
      "C18 UNWINDER STOPPER FORWARD" : Bool;
      "C18 UNWINDER STOPPER BACKWARD" : Bool;
      "C19 UNWINDER DANCER FORWARD" : Bool;
      "C19 UNWINDER DANCER BACKWARD" : Bool;
      "C20 FEEDER CYLINDER DOWN" : Bool;
      "C20 FEEDER CYLINDER UP" : Bool;
      "C21 NG & MANUAL INPUT CYLINDER DOWN" : Bool;
      "C21 NG & MANUAL INPUT CYLINDER UP" : Bool;
      "C22 MAGAZINE LOCK CYLINDER UP" : Bool;
      "C22 MAGAZINE LOCK CYLINDER DOWN" : Bool;
      "C23 VISION PUSHER SUPPORT DOWN" : Bool;
      "C23 VISION PUSHER SUPPORT UP" : Bool;
      "C24 ELECTRODE NG BOX LOCK CYLINDER UP" : Bool;
      "C24 ELECTRODE NG BOX LOCK CYLINDER DOWN" : Bool;
      "C25 FRAME COVER FORWARD" : Bool;
      "C25 FRAME COVER BACKWARD" : Bool;
   END_VAR
BEGIN
END_DATA_BLOCK

DATA_BLOCK "PM05"   // DB271
// stored: MemoryReserve 100
   VAR
      "c1 LEFT UNWINDER EXPEL FORWARD" : Bool;
      "c1 LEFT UNWINDER EXPEL BACKWARD" : Bool;
      SPARE_1 : Bool;
      SPARE_2 : Bool;
      SPARE_3 : Bool;
      SPARE_4 : Bool;
      SPARE_5 : Bool;
      SPARE_6 : Bool;
      SPARE_7 : Bool;
      SPARE_8 : Bool;
      SPARE_9 : Bool;
      SPARE_10 : Bool;
      SPARE_11 : Bool;
      SPARE_12 : Bool;
      SPARE_13 : Bool;
      SPARE_14 : Bool;
   END_VAR
BEGIN
END_DATA_BLOCK

DATA_BLOCK "PM06"   // DB270
// stored: MemoryReserve 100
   VAR
      "c2 RIGHT UNWINDER EXPEL FORWARD" : Bool;
      "c2 RIGHT UNWINDER EXPEL BACKWARD" : Bool;
      SPARE_1 : Bool;
      SPARE_2 : Bool;
      SPARE_3 : Bool;
      SPARE_4 : Bool;
      SPARE_5 : Bool;
      SPARE_6 : Bool;
      SPARE_7 : Bool;
      SPARE_8 : Bool;
      SPARE_9 : Bool;
      SPARE_10 : Bool;
      SPARE_11 : Bool;
      SPARE_12 : Bool;
      SPARE_13 : Bool;
      SPARE_14 : Bool;
   END_VAR
BEGIN
END_DATA_BLOCK

DATA_BLOCK "SBK01"   // DB206
// stored: MemoryReserve 100
   VAR
      "X1-0 No EMG stop: Unwinder" : Bool;
      "X2-1 No EMG stop: Reel cut" : Bool;
      "X3-2 No EMG stop: Vision" : Bool;
      "X4-3 No EMG stop: Conveyor" : Bool;
      "X1-4 reserved" : Bool;
      "X2-5 reserved" : Bool;
      "X3-6 reserved" : Bool;
      "X4-7 reserved" : Bool;
      "X5-0 reserved" : Bool;
      "X6-1 reserved" : Bool;
      "X7-2 reserved" : Bool;
   END_VAR
BEGIN
END_DATA_BLOCK

DATA_BLOCK "SBK02"   // DB208
// stored: MemoryReserve 100
   VAR
      "X1-0 SCS box: SCS mode select, Setup" : Bool;
      "X2-1 SCS box: SCS mode select, Disable" : Bool;
      "X3-2 Frame Corver Detect Sensor" : Bool;
      "X4-3  SAFETY DOOR LOCK7.INPUT" : Bool;
      "X1-4 SCS box: SCS mode select, Auto" : Bool;
      "X2-5 SPARE" : Bool;
      "X3-6 SPARE" : Bool;
      "X4-7 SAFETY DOOR LOCK7.INPUT" : Bool;
      "X5-0 SCS box: Pendant required on, yellow" : Bool;
      "X6-1 SCS box: SCS Disable mode selected, green" : Bool;
      "X7-2 SAFETY DOOR LOCK7.OUTPUT" : Bool;
   END_VAR
BEGIN
END_DATA_BLOCK

DATA_BLOCK "SBK03"   // DB216
// stored: MemoryReserve 100
   VAR
      "X1-0 Roll change LH: Auto" : Bool;
      "X2-1 Roll change RH: Auto" : Bool;
      "X3-2 CART Detect Sensor 1" : Bool;
      "X4-3 CART Detect Sensor 2" : Bool;
      "X1-4 Roll change LH: Change" : Bool;
      "X2-5 Roll change RH: Change" : Bool;
      "X3-6 reserved" : Bool;
      "X4-7 reserved" : Bool;
      "X5-0 Roll change LH: Roll change in progress" : Bool;
      "X6-1 Roll change RH: Roll change in progress" : Bool;
      "X7-2 reserved" : Bool;
   END_VAR
BEGIN
END_DATA_BLOCK

DATA_BLOCK "SBK04"   // DB215
// stored: MemoryReserve 100
   VAR
      "X1-0 Gate EC TOP: Lock" : Bool;
      "X2-1 Gate EC TOP: Reset" : Bool;
      "X3-2 DIFFERENTIAL PRESSURE SWITCH 1 NC" : Bool;
      "X4-3 DIFFERENTIAL PRESSURE SWITCH 2 NC" : Bool;
      "X1-4 Gate EC TOP: Unlock" : Bool;
      "X2-5 reserved" : Bool;
      "X3-6 reserved" : Bool;
      "X4-7 reserved" : Bool;
      "X5-0 Gate EC TOP: Lock lamp on" : Bool;
      "X6-1 Gate EC TOP: Unlock lamp on" : Bool;
      "X7-2 Gate EC TOP: Reset lamp on" : Bool;
   END_VAR
BEGIN
END_DATA_BLOCK

DATA_BLOCK "SBK05"   // DB214
// stored: MemoryReserve 100
   VAR
      "X1-0 Gate EC LH: Lock" : Bool;
      "X2-1 Gate EC LH: Reset" : Bool;
      "X3-2 reserved" : Bool;
      "X4-3 reserved" : Bool;
      "X1-4 Gate EC LH: Unlock" : Bool;
      "X2-5 reserved" : Bool;
      "X3-6 reserved" : Bool;
      "X4-7 reserved" : Bool;
      "X5-0 Gate EC LH: Lock lamp on" : Bool;
      "X6-1 Gate EC LH: Unlock lamp on" : Bool;
      "X7-2 Gate EC LH: Reset lamp on" : Bool;
   END_VAR
BEGIN
END_DATA_BLOCK

DATA_BLOCK "SBK06"   // DB210
// stored: MemoryReserve 100
   VAR
      "X1-0 Gate EC.Top Close" : Bool;
      "X2-1 Gate EC.LH Close" : Bool;
      "X3-2 Gate EC.RH Close" : Bool;
      "X4-3 reserved" : Bool;
      "X1-4 Gate EC.Top Close" : Bool;
      "X2-5 Gate EC.LH Close" : Bool;
      "X3-6 Gate EC.RH Close" : Bool;
      "X4-7 reserved" : Bool;
      "X5-0 Gate EC.Top UnLock" : Bool;
      "X6-1 Gate EC.LH UnLock" : Bool;
      "X7-2 Gate EC.RH UnLock" : Bool;
   END_VAR
BEGIN
END_DATA_BLOCK

DATA_BLOCK "SBK07"   // DB211
// stored: MemoryReserve 100
   VAR
      "X1-0 Gate Cutter Close" : Bool;
      "X2-1 Gate Magazine Close" : Bool;
      "X3-2 Gate Conveyor Close" : Bool;
      "X4-3 reserved" : Bool;
      "X1-4 Gate Cutter Close" : Bool;
      "X2-5 Gate Magazine Close" : Bool;
      "X3-6 Gate Conveyor Close" : Bool;
      "X4-7 reserved" : Bool;
      "X5-0 Gate Cutter Unlock" : Bool;
      "X6-1 Gate Magazine Unlock" : Bool;
      "X7-2 Gate Conveyor Unlock" : Bool;
   END_VAR
BEGIN
END_DATA_BLOCK

DATA_BLOCK "SBK08"   // DB212
// stored: MemoryReserve 100
   VAR
      "X1-0 Gate EC RH: Lock" : Bool;
      "X2-1 Gate EC RH: Reset" : Bool;
      "X3-2 reserved" : Bool;
      "X4-3 reserved" : Bool;
      "X1-4 Gate EC RH: Unlock" : Bool;
      "X2-5 reserved" : Bool;
      "X3-6 reserved" : Bool;
      "X4-7 reserved" : Bool;
      "X5-0 Gate EC RH: Lock lamp on" : Bool;
      "X6-1 Gate EC RH: Unlock lamp on" : Bool;
      "X7-2 Gate EC RH: Reset lamp on" : Bool;
   END_VAR
BEGIN
END_DATA_BLOCK

DATA_BLOCK "SBK09"   // DB209
// stored: MemoryReserve 100
   VAR
      "X1-0 Gate ScrapBox: Lock" : Bool;
      "X2-1 Gate ScrapBox : Reset" : Bool;
      "X3-2 reserved" : Bool;
      "X4-3 reserved" : Bool;
      "X1-4 Gate ScrapBox : Unlock" : Bool;
      "X2-5 reserved" : Bool;
      "X3-6 reserved" : Bool;
      "X4-7 reserved" : Bool;
      "X5-0 Gate ScrapBox : Lock lamp on" : Bool;
      "X6-1 Gate ScrapBox : Unlock lamp on" : Bool;
      "X7-2 Gate ScrapBox : Reset lamp on" : Bool;
   END_VAR
BEGIN
END_DATA_BLOCK

DATA_BLOCK "IdentRfHmi"   // DB213
// stored: MemoryReserve 100
   VAR
      IdentRf : Array[0.."NO_OF_RF_IDENT_DEVICES"] of "typeIdentRf";
      MobileRFID : "LER_typeMobileRFIDInterface";
   END_VAR
BEGIN
END_DATA_BLOCK

ORGANIZATION_BLOCK "Main"   // OB1, LAD, ProgramCycle
TITLE = "Main Program Sweep (Cycle)"
// stored: AutoNumber false, IsIECCheckEnabled true, SetENOAutomatically true
   VAR_INPUT
      Initial_Call : Bool;   // Initial call of this OB
      Remanence : Bool;   // =True, if remanent data are available
   END_VAR
   VAR_TEMP
      tempStart : Bool;
      tempPluse : Bool;
      tempPluse_1 : Bool;
   END_VAR
   VAR CONSTANT
      AlwaysTrue : Bool := TRUE;
   END_VAR
   VAR_TEMP   // added for the SCL form of the ladder/FBD networks
      _w1 : Bool;
      _w2 : Bool;
      _w3 : Bool;
      _w4 : Bool;
   END_VAR
BEGIN

REGION Network 1: First Cycle
   // Set bit to true in first cycle, and false in all other cycles
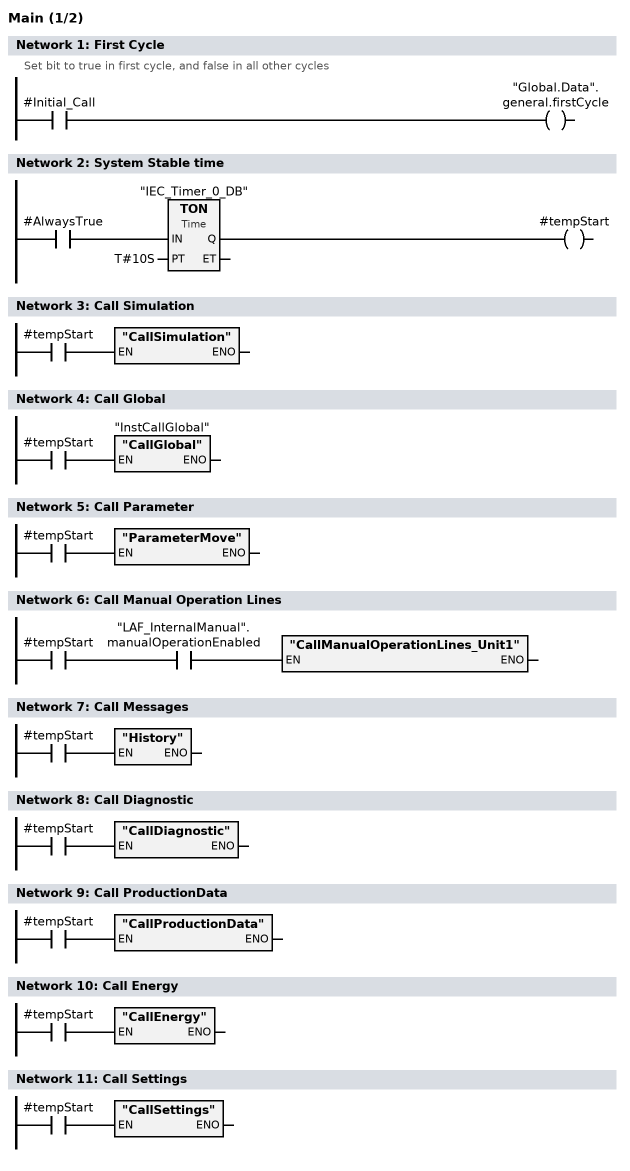
   RUNG wire#powerrail
      Contact( #Initial_Call )
      Coil( "Global.Data".general.firstCycle )
   END_RUNG
   // the same network as SCL:
   "Global.Data".general.firstCycle := #Initial_Call;
END_REGION

REGION Network 2: System Stable time
   RUNG wire#powerrail
      Contact( #AlwaysTrue )
      { S7_Templates := "time_type := Time" } "IEC_Timer_0_DB".TON(pt := T#10S, et =>)
      Coil( #tempStart )
   END_RUNG
   // the same network as SCL:
   "IEC_Timer_0_DB".TON(IN := #AlwaysTrue, PT := T#10S);
   #tempStart := "IEC_Timer_0_DB".Q;
END_REGION

REGION Network 3: Call Simulation
   RUNG wire#powerrail
      Contact( #tempStart )
      "CallSimulation"()
   END_RUNG
   // the same network as SCL:
   IF #tempStart THEN "CallSimulation"(); END_IF;
END_REGION

REGION Network 4: Call Global
   RUNG wire#powerrail
      Contact( #tempStart )
      "InstCallGlobal"()
   END_RUNG
   // the same network as SCL:
   IF #tempStart THEN
       "InstCallGlobal"();   // "CallGlobal"
   END_IF;
END_REGION

REGION Network 5: Call Parameter
   RUNG wire#powerrail
      Contact( #tempStart )
      "ParameterMove"()
   END_RUNG
   // the same network as SCL:
   IF #tempStart THEN "ParameterMove"(); END_IF;
END_REGION

REGION Network 6: Call Manual Operation Lines
   RUNG wire#powerrail
      Contact( #tempStart )
      Contact( "LAF_InternalManual".manualOperationEnabled )
      "CallManualOperationLines_Unit1"()
   END_RUNG
   // the same network as SCL:
   IF #tempStart AND "LAF_InternalManual".manualOperationEnabled THEN
       "CallManualOperationLines_Unit1"();
   END_IF;
END_REGION

REGION Network 7: Call Messages
   RUNG wire#powerrail
      Contact( #tempStart )
      "History"()
   END_RUNG
   // the same network as SCL:
   IF #tempStart THEN "History"(); END_IF;
END_REGION

REGION Network 8: Call Diagnostic
   RUNG wire#powerrail
      Contact( #tempStart )
      "CallDiagnostic"()
   END_RUNG
   // the same network as SCL:
   IF #tempStart THEN "CallDiagnostic"(); END_IF;
END_REGION

REGION Network 9: Call ProductionData
   RUNG wire#powerrail
      Contact( #tempStart )
      "CallProductionData"()
   END_RUNG
   // the same network as SCL:
   IF #tempStart THEN "CallProductionData"(); END_IF;
END_REGION

REGION Network 10: Call Energy
   RUNG wire#powerrail
      Contact( #tempStart )
      "CallEnergy"()
   END_RUNG
   // the same network as SCL:
   IF #tempStart THEN "CallEnergy"(); END_IF;
END_REGION

REGION Network 11: Call Settings
   RUNG wire#powerrail
      Contact( #tempStart )
      "CallSettings"()
   END_RUNG
   // the same network as SCL:
   IF #tempStart THEN "CallSettings"(); END_IF;
END_REGION

REGION Network 12: SinaParaS_SLS Limit Value
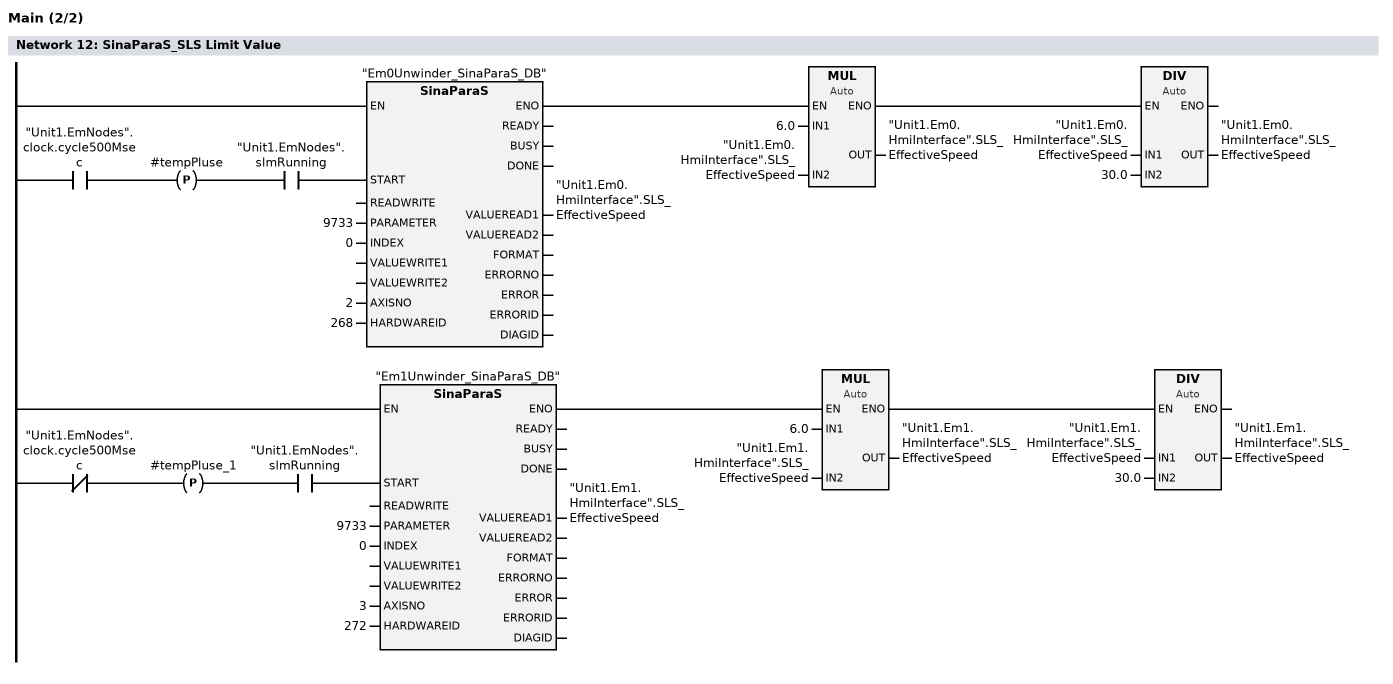
   RUNG wire#powerrail
      "Em0Unwinder_SinaParaS_DB".SinaParaS(Start := wire#w1, ReadWrite :=, Parameter := 9733, Index := 0, ValueWrite1 :=, ValueWrite2 :=, AxisNo := 2, hardwareId := 268, Ready =>, Busy =>, Done =>, ValueRead1 => "Unit1.Em0.HmiInterface".SLS_EffectiveSpeed, ValueRead2 =>, Format =>, ErrorNo =>, Error =>, ErrorId =>, DiagId =>)
      Mul(in1 := 6.0, in2 := "Unit1.Em0.HmiInterface".SLS_EffectiveSpeed, out => "Unit1.Em0.HmiInterface".SLS_EffectiveSpeed)
      Div(in1 := "Unit1.Em0.HmiInterface".SLS_EffectiveSpeed, in2 := 30.0, out => "Unit1.Em0.HmiInterface".SLS_EffectiveSpeed)
   END_RUNG
   RUNG wire#powerrail
      Contact( "Unit1.EmNodes".clock.cycle500Msec )
      P_Trig( #tempPluse )
      Contact( "Unit1.EmNodes".slmRunning )
   END_RUNG wire#w1
   RUNG wire#powerrail
      "Em1Unwinder_SinaParaS_DB".SinaParaS(Start := wire#w2, ReadWrite :=, Parameter := 9733, Index := 0, ValueWrite1 :=, ValueWrite2 :=, AxisNo := 3, hardwareId := 272, Ready =>, Busy =>, Done =>, ValueRead1 => "Unit1.Em1.HmiInterface".SLS_EffectiveSpeed, ValueRead2 =>, Format =>, ErrorNo =>, Error =>, ErrorId =>, DiagId =>)
      Mul(in1 := 6.0, in2 := "Unit1.Em1.HmiInterface".SLS_EffectiveSpeed, out => "Unit1.Em1.HmiInterface".SLS_EffectiveSpeed)
      Div(in1 := "Unit1.Em1.HmiInterface".SLS_EffectiveSpeed, in2 := 30.0, out => "Unit1.Em1.HmiInterface".SLS_EffectiveSpeed)
   END_RUNG
   RUNG wire#powerrail
      I_Contact( "Unit1.EmNodes".clock.cycle500Msec )
      P_Trig( #tempPluse_1 )
      Contact( "Unit1.EmNodes".slmRunning )
   END_RUNG wire#w2
   // the same network as SCL:
   #_w1 := "Unit1.EmNodes".clock.cycle500Msec AND NOT #tempPluse;   // rising edge
   #tempPluse := "Unit1.EmNodes".clock.cycle500Msec;
   "Em0Unwinder_SinaParaS_DB"(Start := #_w1 AND "Unit1.EmNodes".slmRunning,   // SinaParaS
                           Parameter := 9733,
                           Index := 0,
                           AxisNo := 2,
                           hardwareId := 268,
                           ValueRead1 => "Unit1.Em0.HmiInterface".SLS_EffectiveSpeed,
                           ENO => #_w2);
   IF #_w2 THEN
       "Unit1.Em0.HmiInterface".SLS_EffectiveSpeed := 6.0 * "Unit1.Em0.HmiInterface".SLS_EffectiveSpeed;
       "Unit1.Em0.HmiInterface".SLS_EffectiveSpeed := "Unit1.Em0.HmiInterface".SLS_EffectiveSpeed / 30.0;
   END_IF;
   #_w3 := NOT "Unit1.EmNodes".clock.cycle500Msec AND NOT #tempPluse_1;   // rising edge
   #tempPluse_1 := NOT "Unit1.EmNodes".clock.cycle500Msec;
   "Em1Unwinder_SinaParaS_DB"(Start := #_w3 AND "Unit1.EmNodes".slmRunning,   // SinaParaS
                           Parameter := 9733,
                           Index := 0,
                           AxisNo := 3,
                           hardwareId := 272,
                           ValueRead1 => "Unit1.Em1.HmiInterface".SLS_EffectiveSpeed,
                           ENO => #_w4);
   IF #_w4 THEN
       "Unit1.Em1.HmiInterface".SLS_EffectiveSpeed := 6.0 * "Unit1.Em1.HmiInterface".SLS_EffectiveSpeed;
       "Unit1.Em1.HmiInterface".SLS_EffectiveSpeed := "Unit1.Em1.HmiInterface".SLS_EffectiveSpeed / 30.0;
   END_IF;
END_REGION
END_ORGANIZATION_BLOCK

FUNCTION "CallSimulation" : Void   // FC22, LAD
TITLE = CallSimulation
// This blocks switches between simulation with SIMIT and PLCSIM Advanced or with PLCSIM and PLC internal simulation function blocks
// stored: IsIECCheckEnabled true, SetENOAutomatically true
   VAR CONSTANT
      True : Bool := true;   // OEM: replace with ProDiag statuses that command unit state
      False : Bool;
   END_VAR
   VAR_TEMP   // added for the SCL form of the ladder/FBD networks
      _w1 : Bool;
      _w2 : Bool;
      _w3 : Bool;
      _w4 : Bool;
      _w5 : Bool;
   END_VAR
BEGIN

REGION Network 1: SIMIT simulation currently running
   // The input "0.000CC1-KE50_I1.6_SimitRunning" is a life bit from SIMIT, which is always TRUE while SIMIT is running. The following actions are performed in that case:
   // - Simulation button in HMI is not shown when a SIMIT simulation is currently running
   // - Deactivate PLC internal simulation while SIMIT simulation is running
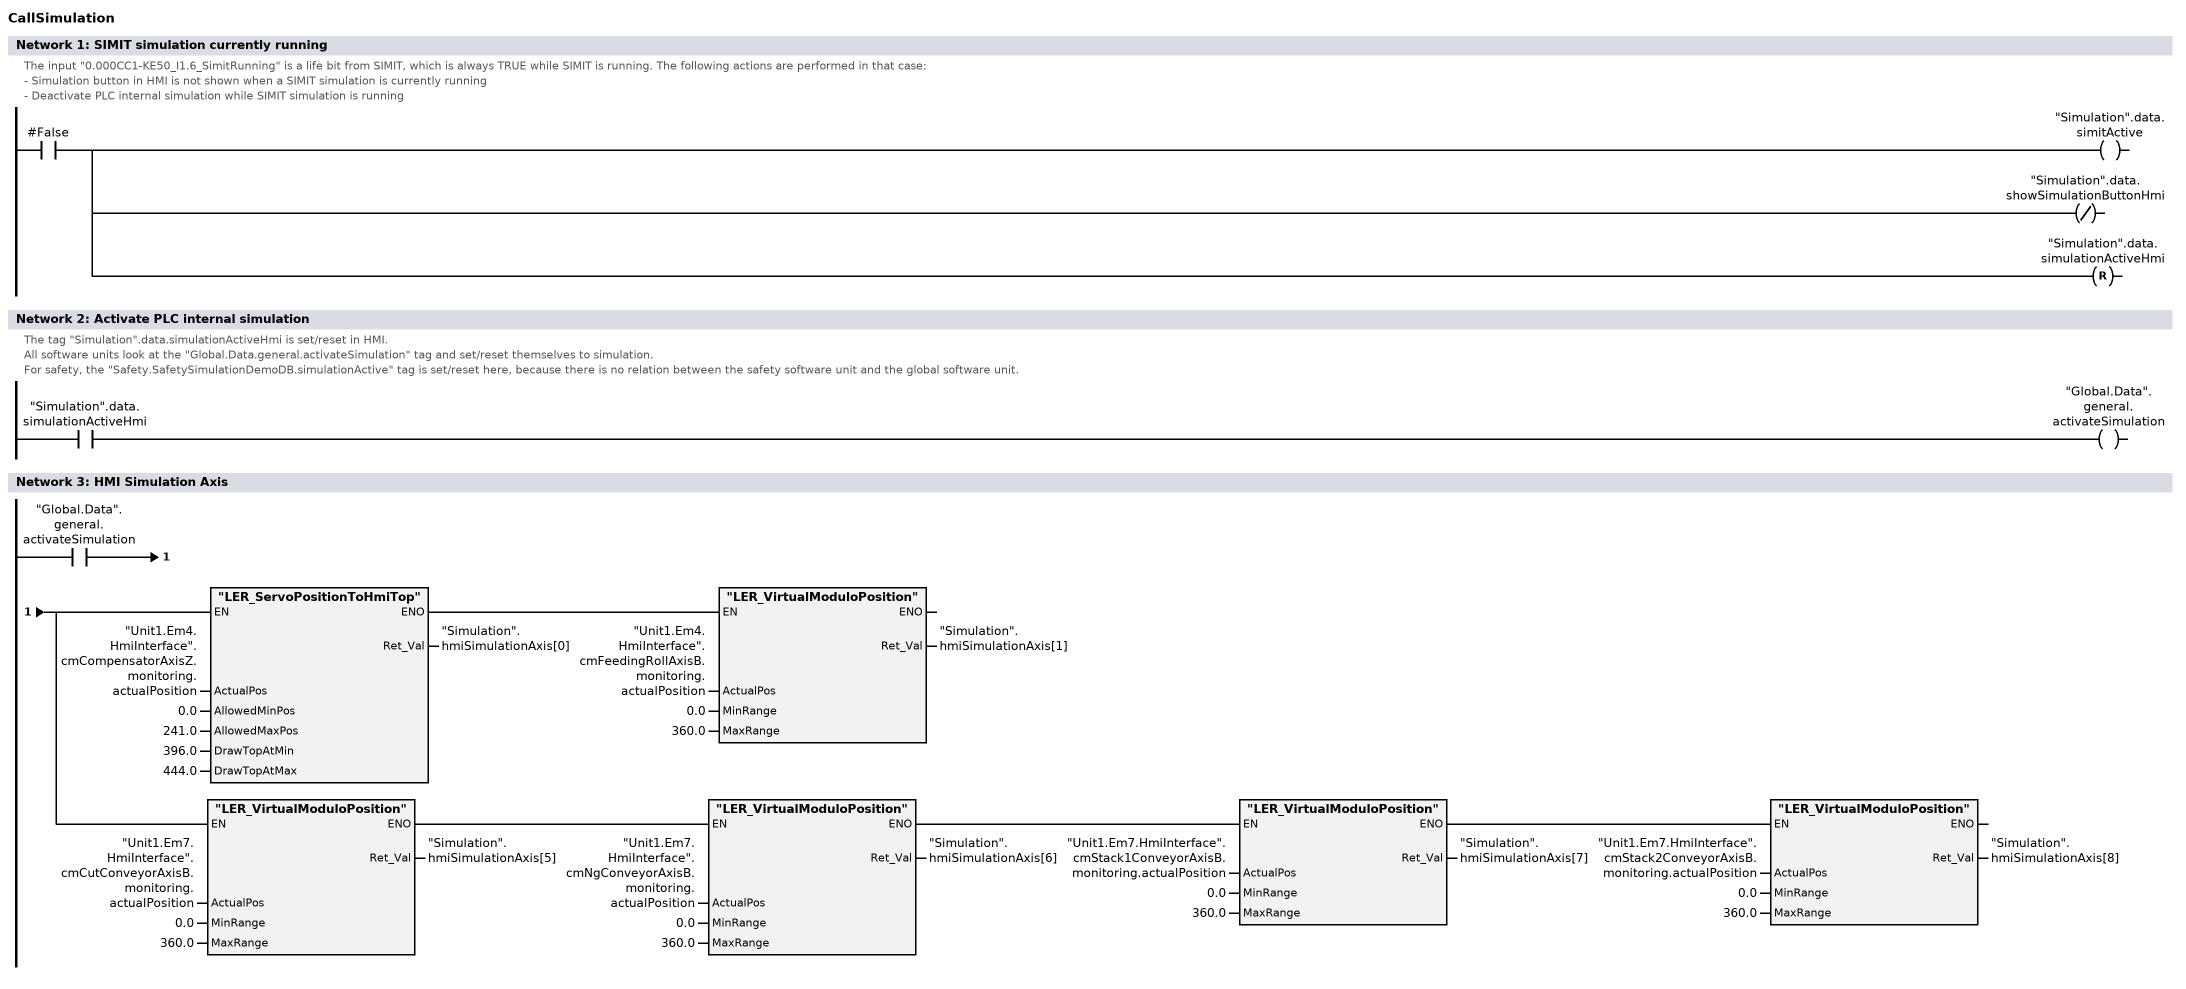
   RUNG wire#powerrail
      Contact( #False )
      wire#w1
      Coil( "Simulation".data.simitActive )
   END_RUNG
   RUNG wire#w1
      I_Coil( "Simulation".data.showSimulationButtonHmi )
   END_RUNG
   RUNG wire#w1
      R_Coil( "Simulation".data.simulationActiveHmi )
   END_RUNG
   // the same network as SCL:
   "Simulation".data.simitActive := #False;
   "Simulation".data.showSimulationButtonHmi := NOT #False;
   IF #False THEN "Simulation".data.simulationActiveHmi := FALSE; END_IF;
END_REGION

REGION Network 2: Activate PLC internal simulation
   // The tag "Simulation".data.simulationActiveHmi is set/reset in HMI.
   // 
   // All software units look at the "Global.Data.general.activateSimulation" tag and set/reset themselves to simulation.
   // 
   // For safety, the "Safety.SafetySimulationDemoDB.simulationActive" tag is set/reset here, because there is no relation between the safety software unit and the global software unit.
   RUNG wire#powerrail
      Contact( "Simulation".data.simulationActiveHmi )
      Coil( "Global.Data".general.activateSimulation )
   END_RUNG
   // the same network as SCL:
   "Global.Data".general.activateSimulation := "Simulation".data.simulationActiveHmi;
END_REGION

REGION Network 3: HMI Simulation Axis
   RUNG wire#powerrail
      Contact( "Global.Data".general.activateSimulation )
      wire#w1
      "LER_ServoPositionToHmiTop"(ActualPos := "Unit1.Em4.HmiInterface".cmCompensatorAxisZ.monitoring.actualPosition, AllowedMinPos := 0.0, AllowedMaxPos := 241.0, DrawTopAtMin := 396.0, DrawTopAtMax := 444.0, Ret_Val => "Simulation".hmiSimulationAxis[0])
      "LER_VirtualModuloPosition"(ActualPos := "Unit1.Em4.HmiInterface".cmFeedingRollAxisB.monitoring.actualPosition, MinRange := 0.0, MaxRange := 360.0, Ret_Val => "Simulation".hmiSimulationAxis[1])
   END_RUNG
   RUNG wire#w1
      "LER_VirtualModuloPosition"(ActualPos := "Unit1.Em7.HmiInterface".cmCutConveyorAxisB.monitoring.actualPosition, MinRange := 0.0, MaxRange := 360.0, Ret_Val => "Simulation".hmiSimulationAxis[5])
      "LER_VirtualModuloPosition"(ActualPos := "Unit1.Em7.HmiInterface".cmNgConveyorAxisB.monitoring.actualPosition, MinRange := 0.0, MaxRange := 360.0, Ret_Val => "Simulation".hmiSimulationAxis[6])
      "LER_VirtualModuloPosition"(ActualPos := "Unit1.Em7.HmiInterface".cmStack1ConveyorAxisB.monitoring.actualPosition, MinRange := 0.0, MaxRange := 360.0, Ret_Val => "Simulation".hmiSimulationAxis[7])
      "LER_VirtualModuloPosition"(ActualPos := "Unit1.Em7.HmiInterface".cmStack2ConveyorAxisB.monitoring.actualPosition, MinRange := 0.0, MaxRange := 360.0, Ret_Val => "Simulation".hmiSimulationAxis[8])
   END_RUNG
   // the same network as SCL:
   #_w2 := "Global.Data".general.activateSimulation;
   "Simulation".hmiSimulationAxis[0] := "LER_ServoPositionToHmiTop"(EN := "Global.Data".general.activateSimulation,
                           ActualPos := "Unit1.Em4.HmiInterface".cmCompensatorAxisZ.monitoring.actualPosition,
                           AllowedMinPos := 0.0,
                           AllowedMaxPos := 241.0,
                           DrawTopAtMin := 396.0,
                           DrawTopAtMax := 444.0,
                           ENO => #_w1);
   IF #_w1 THEN
       "Simulation".hmiSimulationAxis[1] := "LER_VirtualModuloPosition"(ActualPos := "Unit1.Em4.HmiInterface".cmFeedingRollAxisB.monitoring.actualPosition,
                               MinRange := 0.0,
                               MaxRange := 360.0);
   END_IF;
   "Simulation".hmiSimulationAxis[5] := "LER_VirtualModuloPosition"(EN := #_w2,
                           ActualPos := "Unit1.Em7.HmiInterface".cmCutConveyorAxisB.monitoring.actualPosition,
                           MinRange := 0.0,
                           MaxRange := 360.0,
                           ENO => #_w3);
   "Simulation".hmiSimulationAxis[6] := "LER_VirtualModuloPosition"(EN := #_w3,
                           ActualPos := "Unit1.Em7.HmiInterface".cmNgConveyorAxisB.monitoring.actualPosition,
                           MinRange := 0.0,
                           MaxRange := 360.0,
                           ENO => #_w4);
   "Simulation".hmiSimulationAxis[7] := "LER_VirtualModuloPosition"(EN := #_w4,
                           ActualPos := "Unit1.Em7.HmiInterface".cmStack1ConveyorAxisB.monitoring.actualPosition,
                           MinRange := 0.0,
                           MaxRange := 360.0,
                           ENO => #_w5);
   IF #_w5 THEN
       "Simulation".hmiSimulationAxis[8] := "LER_VirtualModuloPosition"(ActualPos := "Unit1.Em7.HmiInterface".cmStack2ConveyorAxisB.monitoring.actualPosition,
                               MinRange := 0.0,
                               MaxRange := 360.0);
   END_IF;
END_REGION
END_FUNCTION

FUNCTION_BLOCK "CallGlobal"   // FB48, LAD
TITLE = CallGlobal
// All blocks that provide data to the DB Global.Data are called here. That includes blocks to generate system data as well as blocks that connect handle multiple HMIs.
// stored: IsIECCheckEnabled true, MemoryReserve 100, SetENOAutomatically true
   VAR
      statClockSysMemOld { ExternalWritable := 'False'} : Byte;   // Old value system memory evaluation
      statPulse : Array[0..9] of Bool;
      instLAF_PowerOnOff { ExternalWritable := 'False'} : "LAF_PowerOnOff";
      instLAF_HmiHeaderManager { ExternalWritable := 'False'} : "LAF_HmiHeaderManager";
      instLAF_ClockGen { ExternalWritable := 'False'} : "LAF_ClockGenerator";
      instLSNTP_Server { ExternalWritable := 'False'} : "LSNTP_Server";
      statTonTimer { ExternalWritable := 'False'} : Array[0..9] of TON_TIME;
   END_VAR
   VAR_TEMP
      tempIndex : DInt;   // Temp variable for for loop
      tempAcknowledge : Bool;   // Summarized acknowledge command
      tempPowerOff : Bool;   // Summarized power off command
      tempPowerOn : Bool;   // Summarized power on command
      tempPowerStatus : Int;   // 0 - Off, 1 - Paused, 2 - On
      tempResultXor : Byte;   // Interim result of XOR operation
      tempPosPulse : Byte;   // Interim result puls calculation
      temp_REPLACE_THIS : HW_ANY;
   END_VAR
   VAR CONSTANT
      RESET_BUTTON__COULD_BE_ADDED_HERE : Bool := false;   // Placeholder for a potential global reset button
      TRUE : Bool := TRUE;
      FALSE : Bool := FALSE;
   END_VAR
   VAR_TEMP   // added for the SCL form of the ladder/FBD networks
      _w1 : Bool;
      _w2 : Bool;
      _w3 : Bool;
      _w4 : Bool;
      _w5 : Bool;
      _w6 : Bool;
      _w7 : Bool;
      _w8 : Bool;
   END_VAR
BEGIN

REGION Network 1 (SCL): Summarize HMI commands
   // Read commands for acknowledge, powerOn and powerOff from the different HMI panels and summarize them in temp variables for further logic in this block.
   // Initialize temp variables
   #tempAcknowledge :=
   #tempPowerOff :=
   #tempPowerOn := FALSE;

   // Loop through the HMI panels and summarize the commands
   FOR #tempIndex := 0 TO "NO_OF_PANELS" DO
       #tempAcknowledge := #tempAcknowledge OR "Hmi".mainHeader[#tempIndex].hmiToPlc.acknowledge;
       #tempPowerOff := #tempPowerOff OR "Hmi".mainHeader[#tempIndex].hmiToPlc.powerCommands.%X0;
       #tempPowerOn := #tempPowerOn OR "Hmi".mainHeader[#tempIndex].hmiToPlc.powerCommands.%X1;
   END_FOR;
END_REGION

REGION Network 2: Global Acknowledge
   // The global acknowledge command from the hmi button is assigned to Global.Data.general.acknowledge: This bit it forwarded to all underlaying modules
   // If a hard-wired global reset button exists, it can
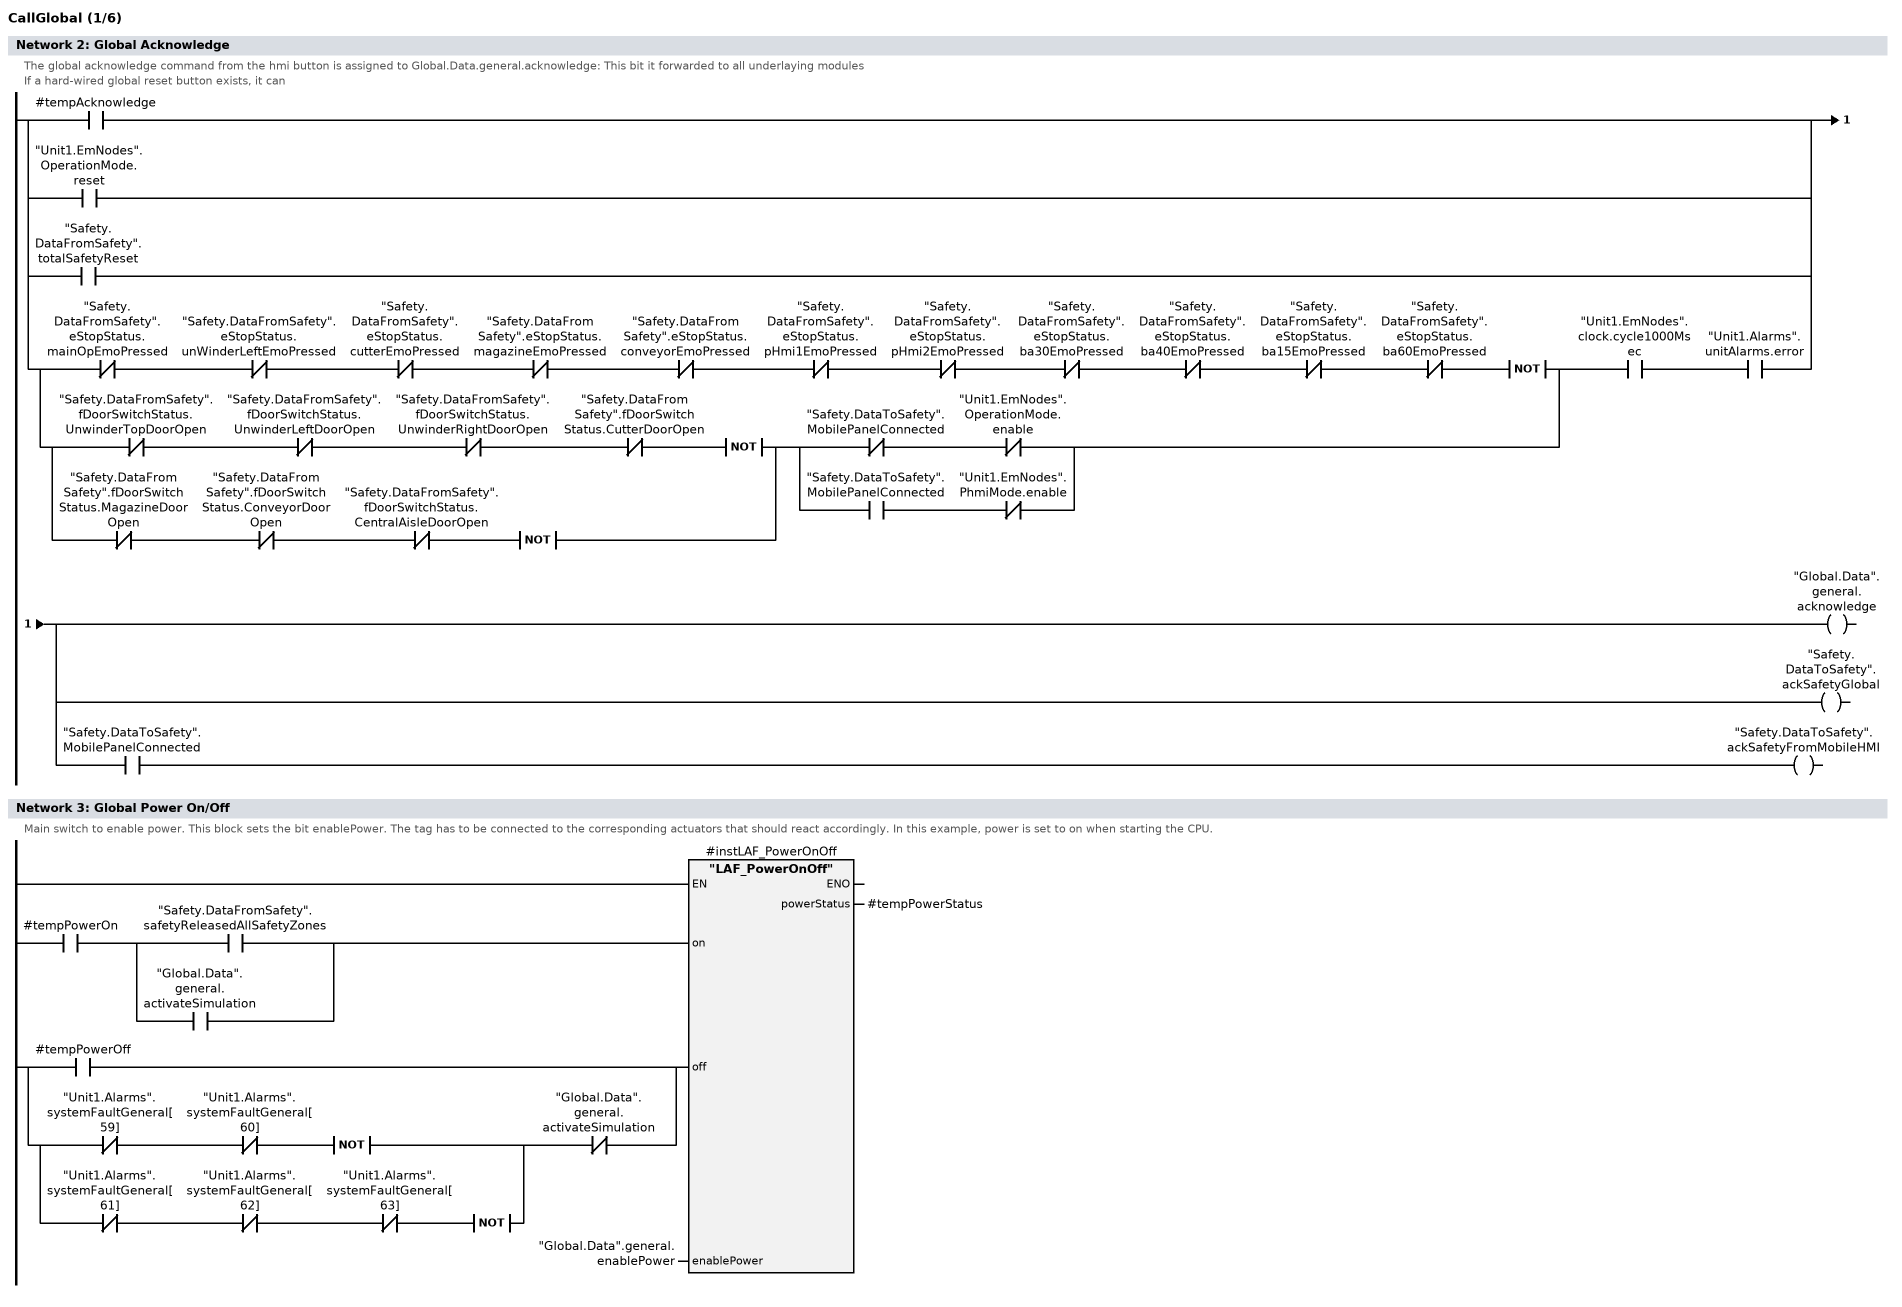
   RUNG wire#powerrail
      Contact( #tempAcknowledge )
      wire#w1
      Coil( "Global.Data".general.acknowledge )
   END_RUNG
   RUNG wire#powerrail
      Contact( "Unit1.EmNodes".OperationMode.reset )
   END_RUNG wire#w1
   RUNG wire#powerrail
      Contact( "Safety.DataFromSafety".totalSafetyReset )
   END_RUNG wire#w1
   RUNG wire#powerrail
      I_Contact( "Safety.DataFromSafety".eStopStatus.mainOpEmoPressed )
      I_Contact( "Safety.DataFromSafety".eStopStatus.unWinderLeftEmoPressed )
      I_Contact( "Safety.DataFromSafety".eStopStatus.cutterEmoPressed )
      I_Contact( "Safety.DataFromSafety".eStopStatus.magazineEmoPressed )
      I_Contact( "Safety.DataFromSafety".eStopStatus.conveyorEmoPressed )
      I_Contact( "Safety.DataFromSafety".eStopStatus.pHmi1EmoPressed )
      I_Contact( "Safety.DataFromSafety".eStopStatus.pHmi2EmoPressed )
      I_Contact( "Safety.DataFromSafety".eStopStatus.ba30EmoPressed )
      I_Contact( "Safety.DataFromSafety".eStopStatus.ba40EmoPressed )
      I_Contact( "Safety.DataFromSafety".eStopStatus.ba15EmoPressed )
      I_Contact( "Safety.DataFromSafety".eStopStatus.ba60EmoPressed )
      Not()
      wire#w2
      Contact( "Unit1.EmNodes".clock.cycle1000Msec )
      Contact( "Unit1.Alarms".unitAlarms.error )
   END_RUNG wire#w1
   RUNG wire#powerrail
      I_Contact( "Safety.DataFromSafety".fDoorSwitchStatus.UnwinderTopDoorOpen )
      I_Contact( "Safety.DataFromSafety".fDoorSwitchStatus.UnwinderLeftDoorOpen )
      I_Contact( "Safety.DataFromSafety".fDoorSwitchStatus.UnwinderRightDoorOpen )
      I_Contact( "Safety.DataFromSafety".fDoorSwitchStatus.CutterDoorOpen )
      Not()
      wire#w3
      I_Contact( "Safety.DataToSafety".MobilePanelConnected )
      I_Contact( "Unit1.EmNodes".OperationMode.enable )
   END_RUNG wire#w2
   RUNG wire#powerrail
      I_Contact( "Safety.DataFromSafety".fDoorSwitchStatus.MagazineDoorOpen )
      I_Contact( "Safety.DataFromSafety".fDoorSwitchStatus.ConveyorDoorOpen )
      I_Contact( "Safety.DataFromSafety".fDoorSwitchStatus.CentralAisleDoorOpen )
      Not()
   END_RUNG wire#w3
   RUNG wire#w3
      Contact( "Safety.DataToSafety".MobilePanelConnected )
      I_Contact( "Unit1.EmNodes".PhmiMode.enable )
   END_RUNG wire#w2
   RUNG wire#w1
      Coil( "Safety.DataToSafety".ackSafetyGlobal )
   END_RUNG
   RUNG wire#w1
      Contact( "Safety.DataToSafety".MobilePanelConnected )
      Coil( "Safety.DataToSafety".ackSafetyFromMobileHMI )
   END_RUNG
   // the same network as SCL:
   "Global.Data".general.acknowledge := #tempAcknowledge OR "Unit1.EmNodes".OperationMode.reset OR "Safety.DataFromSafety".totalSafetyReset OR ((NOT (NOT "Safety.DataFromSafety".eStopStatus.mainOpEmoPressed AND NOT "Safety.DataFromSafety".eStopStatus.unWinderLeftEmoPressed AND NOT "Safety.DataFromSafety".eStopStatus.cutterEmoPressed AND NOT "Safety.DataFromSafety".eStopStatus.magazineEmoPressed AND NOT "Safety.DataFromSafety".eStopStatus.conveyorEmoPressed AND NOT "Safety.DataFromSafety".eStopStatus.pHmi1EmoPressed AND NOT "Safety.DataFromSafety".eStopStatus.pHmi2EmoPressed AND NOT "Safety.DataFromSafety".eStopStatus.ba30EmoPressed AND NOT "Safety.DataFromSafety".eStopStatus.ba40EmoPressed AND NOT "Safety.DataFromSafety".eStopStatus.ba15EmoPressed AND NOT "Safety.DataFromSafety".eStopStatus.ba60EmoPressed) OR ((NOT (NOT "Safety.DataFromSafety".fDoorSwitchStatus.UnwinderTopDoorOpen AND NOT "Safety.DataFromSafety".fDoorSwitchStatus.UnwinderLeftDoorOpen AND NOT "Safety.DataFromSafety".fDoorSwitchStatus.UnwinderRightDoorOpen AND NOT "Safety.DataFromSafety".fDoorSwitchStatus.CutterDoorOpen) OR NOT (NOT "Safety.DataFromSafety".fDoorSwitchStatus.MagazineDoorOpen AND NOT "Safety.DataFromSafety".fDoorSwitchStatus.ConveyorDoorOpen AND NOT "Safety.DataFromSafety".fDoorSwitchStatus.CentralAisleDoorOpen)) AND ((NOT "Safety.DataToSafety".MobilePanelConnected AND NOT "Unit1.EmNodes".OperationMode.enable) OR ("Safety.DataToSafety".MobilePanelConnected AND NOT "Unit1.EmNodes".PhmiMode.enable)))) AND "Unit1.EmNodes".clock.cycle1000Msec AND "Unit1.Alarms".unitAlarms.error);
   "Safety.DataToSafety".ackSafetyGlobal := "Global.Data".general.acknowledge;
   "Safety.DataToSafety".ackSafetyFromMobileHMI := "Global.Data".general.acknowledge AND "Safety.DataToSafety".MobilePanelConnected;
END_REGION

REGION Network 3: Global Power On/Off
   // Main switch to enable power. This block sets the bit enablePower. The tag has to be connected to the corresponding actuators that should react accordingly. In this example, power is set to on when starting the CPU.
   RUNG wire#powerrail
      #instLAF_PowerOnOff(on := wire#w2, off := wire#w4, enablePower := "Global.Data".general.enablePower, powerStatus => #tempPowerStatus)
   END_RUNG
   RUNG wire#powerrail
      Contact( #tempPowerOn )
      wire#w1
      Contact( "Safety.DataFromSafety".safetyReleasedAllSafetyZones )
   END_RUNG wire#w2
   RUNG wire#w1
      Contact( "Global.Data".general.activateSimulation )
   END_RUNG wire#w2
   RUNG wire#powerrail
      Contact( #tempPowerOff )
   END_RUNG wire#w4
   RUNG wire#powerrail
      I_Contact( "Unit1.Alarms".systemFaultGeneral[59] )
      I_Contact( "Unit1.Alarms".systemFaultGeneral[60] )
      Not()
      wire#w3
      I_Contact( "Global.Data".general.activateSimulation )
   END_RUNG wire#w4
   RUNG wire#powerrail
      I_Contact( "Unit1.Alarms".systemFaultGeneral[61] )
      I_Contact( "Unit1.Alarms".systemFaultGeneral[62] )
      I_Contact( "Unit1.Alarms".systemFaultGeneral[63] )
      Not()
   END_RUNG wire#w3
   // the same network as SCL:
   #instLAF_PowerOnOff(on := #tempPowerOn AND ("Safety.DataFromSafety".safetyReleasedAllSafetyZones OR "Global.Data".general.activateSimulation),   // "LAF_PowerOnOff"
                       off := #tempPowerOff OR ((NOT (NOT "Unit1.Alarms".systemFaultGeneral[59] AND NOT "Unit1.Alarms".systemFaultGeneral[60]) OR NOT (NOT "Unit1.Alarms".systemFaultGeneral[61] AND NOT "Unit1.Alarms".systemFaultGeneral[62] AND NOT "Unit1.Alarms".systemFaultGeneral[63])) AND NOT "Global.Data".general.activateSimulation),
                       enablePower := "Global.Data".general.enablePower,
                       powerStatus => #tempPowerStatus);
END_REGION

REGION Network 4 (SCL): Write power status to HMI panels
   // Write power status back to all connected HMI panels
   // Loop through the panels and set the power status
   FOR #tempIndex := 0 TO "NO_OF_PANELS" DO
       "Hmi".mainHeader[#tempIndex].plcToHmi.powerStatus := #tempPowerStatus;
   END_FOR;
END_REGION

